// TwinCAT 3 PLC project PMPS
// Title: PMPS
// Company: SLAC - LCLS
// Author: Alex Wallace and contributors
// ProjectVersion: 0.0.0
// Description: Collection of PMPS functionality for LCLS PLCs
// ProgramVersion: 3.1.4023.0
// CompilerDefines: L
// libraries:
//   LCLS General, * (SLAC)
//   Tc2_MC2, * (Beckhoff Automation GmbH)
//   Tc2_Standard, * (Beckhoff Automation GmbH)
//   Tc2_System, * (Beckhoff Automation GmbH)
//   Tc2_Utilities, * (Beckhoff Automation GmbH)
//   Tc3_JsonXml, * (Beckhoff Automation GmbH)
//   Tc3_Module, * (Beckhoff Automation GmbH)
//   TcUnit,1.2.0.0,www.tcunit.org
// project tree:
//   AncillaryComponents/ FB_JsonDocToSafeBP.TcPOU, FB_JsonFileToJsonDoc.TcPOU, FB_TempSensor_FFO.TcPOU, FB_PressSensor_FFO.TcPOU
//   DUTs/InternalDUT/ E_MPSBeamRates.TcDUT, E_MPSBeamClasses.TcDUT, K_Apertures.TcDUT, K_Attenuators.TcDUT, K_Stopper.TcDUT, L_Apertures.TcDUT, L_Attenuators.TcDUT, L_Stopper.TcDUT, ST_AttenuatorStatus.TcDUT, ST_BP_ArbInternal.TcDUT, ST_FF.TcDUT, ST_FFInfo.TcDUT, ST_FFOverride.TcDUT, ST_PMPS_Aperture.TcDUT, ST_PMPS_Attenuator.TcDUT, T_HashTableEntry.TcDUT
//   DUTs/ PMPS_CODES.TcDUT, ST_DeviceState.TcDUT, ST_DeviceStateExt.TcDUT, ST_DeviceStateTable.TcDUT
//   DUTs/UserDUT/ E_BridgeLinkStatus.TcDUT, E_BridgeStatus.TcDUT, E_DataStatus.TcDUT, E_EcCommState.TcDUT, ST_ReactiveParams.TcDUT, ST_BeamParams.TcDUT, ST_DbStateParams.TcDUT, ST_Device.TcDUT
//   GVLs/ PMPS_GVL.TcGVL, PMPS_PARAM.TcGVL, PMPS_TOOLS.TcGVL
//   HelperFunctions/ FB_DummyHA.TcPOU, FB_DummyArbIO.TcPOU, F_BPWithID.TcPOU, F_DifferentBeamParams.TcPOU, F_eVExcludeRange.TcPOU, F_eVIncludeRange.TcPOU, F_eVRangeCalculator.TcPOU, F_eVWithinSpec.TcPOU, F_InitTestBP.TcPOU, F_SafeBPCompare.TcPOU, F_SafeBPCompare0Rate.TcPOU, F_SetBeamParams.TcPOU, F_SetGoodAttStatus.TcPOU, F_SetStateParams.TcPOU, F_PMPS_JSON.TcPOU, F_ValidReqID.TcPOU, PE_Ranges.TcPOU, F_AttenuatorOK.TcPOU
//   HelperFunctions/TypeTranslators/ APT_TO_IO.TcPOU, ATT_TO_IO.TcPOU, BP_TO_IO.TcPOU, F_DeviceState_To_DeviceStateExt.TcPOU, IO_TO_APT.TcPOU, IO_TO_ATT.TcPOU, IO_TO_BP.TcPOU
//   ImplicitChecks/ CheckBounds.TcPOU, CheckDivDInt.TcPOU, CheckDivLInt.TcPOU, CheckDivLReal.TcPOU, CheckDivReal.TcPOU, CheckLRangeSigned.TcPOU, CheckLRangeUnsigned.TcPOU, CheckPointer.TcPOU, CheckRangeSigned.TcPOU, CheckRangeUnsigned.TcPOU
//   / MAIN.TcPOU, PlcTask.TcTTO
//   MajorComponents/Arbiter/ FB_VetoArbiter.TcPOU, FB_Arbiter.TcPOU, FB_BeamParamAssertionPool.TcPOU
//   MajorComponents/BPTM/ BeamParameterTransitionManager.TcPOU, E_BPTMState.TcDUT
//   MajorComponents/ FB_BPControlDevice.TcPOU, FB_RateFromEPICS.TcPOU, FB_BeamClassFromEPICS.TcPOU, I_LowerAuthority.TcIO, I_UndulatorComplex.TcIO, FB_BPRequestor.TcPOU, FB_LinearDeviceStateTable.TcPOU, FB_LinearGovernor.TcPOU, I_HigherAuthority.TcIO
//   MajorComponents/PhotonEnergyInterface/ FB_AcceleratorLinks.TcPOU, FB_Hgvpu.TcPOU, FB_LPhotonEnergy.TcPOU, FB_KPhotonEnergy.TcPOU, FB_PhotonEnergy.TcPOU, FB_SXU.TcPOU, FB_UndulatorSegment.TcPOU, F_CalculatePhotonEnergy.TcPOU
//   MajorComponents/FastFaults/ FB_FastFault.TcPOU, FB_HardwareFFOutput.TcPOU
//   MajorComponents/InterPlcComm/ FB_ArbiterToSubSys_IO.TcPOU, FB_BridgeDiagnostics.TcPOU, FB_SubSysToArbiter_IO.TcPOU
//   MajorComponents/InterPlcComm/Sanitization/ I_FallibleLreal.TcIO, FB_FallibleRealFromEtherCAT.TcPOU
//   MajorComponents/PMPS_MPS_Interface/ FB_BeamClassOutputs.TcPOU, FB_BeamClassOutputs_BCD.TcPOU, FB_CTLS_Outputs.TcPOU, FB_MachineModeFromEPICS.TcPOU, FB_PhotonEnergyWatcher.TcPOU, FB_BeamClassWatcher.TcPOU
//   MajorComponents/SimulationFB/ FB_eVSimulator.TcPOU, FB_MachineSimulator.TcPOU
//   MajorComponents/Stoppers/ FB_KStopper.TcPOU, FB_KVetoDevice.TcPOU, FB_LVetoDevice.TcPOU, FB_LStopper.TcPOU, FB_StopperWatcher.TcPOU, FB_VetoDevice.TcPOU
//   TestComponents/DUT/ E_ArbDosTestStates.TcDUT, E_BPTMTestStates.TcDUT
//   TestComponents/ FB_Arbiter_Test.TcPOU, FB_VetoArbiter_Test.TcPOU, FB_AttenuatorSimulator.TcPOU, FB_BPTM_Test.TcPOU, FB_ArbToSubsys_Test.TcPOU, FB_DiffBP_Test.TcPOU, FB_SubsysToArb_Test.TcPOU, FB_evRangeCalculator_Test.TcPOU, FB_eVWithinSpec_Test.TcPOU, FB_FastFault_Test.TcPOU, FB_PhotonEnergyWatcher_Test.TcPOU, FB_SafeBPCompare_Test.TcPOU, FB_SolidAttenuator.TcPOU (excluded from build)
// real-time tasks:
//   TASK PlcTask: cycle T#10ms, priority 20, ADS port 350

CONFIGURATION PMPS
    RESOURCE PLC ON TwinCAT3
        TASK PlcTask(INTERVAL := T#10ms, PRIORITY := 20);
        PROGRAM MAIN WITH PlcTask : MAIN;
    END_RESOURCE
END_CONFIGURATION

// ---- DUTs/InternalDUT/E_MPSBeamRates.TcDUT

TYPE E_MPSBeamRates :
(
    MPSRateInvalid            :=  0,
    MPSRate0Hz                :=  1,
    (* Previously used 2 and 3 for single shot and burst *)
    MPSRate1Hz                :=  4,
    MPSRate10Hz               :=  5,
    MPSRate30Hz               :=  6,
    MPSRate60Hz               :=  7,
    MPSRate120Hz              :=  8,
    MPSRateUnknown            :=  9,
    MPSRateSingleShot         := 10,
    MPSRateBurstMode          := 11,
    MPSRateBurstModeNotActive := 12,
    MPSNumberOfBeamRates      := 13,
    MPSRateBurstInvalid       := 14
)UINT;
END_TYPE

// ---- DUTs/InternalDUT/E_MPSBeamClasses.TcDUT

TYPE E_MPSBeamClasses :
(
    Beam_Off    :=  0,
    Kicker_STBY :=  1,
    BC1Hz       :=  2,
    BC10Hz      :=  3,
    BC120Hz     :=  4,
    Diagnostic  :=  5,
    Tuning      :=  6,
    MAP_1       :=  7,
    MAP_5       :=  8,
    MAP_10      :=  9,
    MAP_25      := 10,
    MAP_50      := 11,
    MAP_100     := 12,
    FULL        := 13,
    SPARE1      := 14,
    SPARE2      := 15
);
END_TYPE

// ---- DUTs/InternalDUT/K_Apertures.TcDUT
{attribute 'qualified_only'}
{attribute 'strict'}
{attribute 'to_string'}
TYPE K_Apertures :
(
    SL1K0 := 1,
    SL2K0 := 2
);
END_TYPE

// ---- DUTs/InternalDUT/K_Attenuators.TcDUT
{attribute 'qualified_only'}
{attribute 'strict'}
TYPE K_Attenuators :
(
    AT1K0 := 1, // FEE Gas Attenuator
    AT1K4 := 2, // TMO Solid Attenuator in the FEE
    AT1K2 := 3, // RIX Solid Attenuator
    AT2K2 := 4, // RIX Solid Attenuator
    AT1K3 := 5 // TXI Solid Attenuator
);
END_TYPE

// ---- DUTs/InternalDUT/K_Stopper.TcDUT
{attribute 'qualified_only'}
{attribute 'strict'}
TYPE K_Stopper :
(
    ST3K4 := 1, // TMO PPS stopper in
    ST1K2 := 2, // RIX PPS stopper in
    MR1K1_IN := 3, // Monochromator focus optic vertical state
    MR1K1_OUT := 4, // Monochromator focus optic vertical state
    MR1K3_IN := 5, // TXI MR1K3 Offset Mirror horizontal state
    MR1K3_OUT := 6, // TXI MR1K3 Offset Mirror horizontal state
    ST4K4 := 7, //TMO ST4K4 Photon Terminator In Limit Switch
    ST1K0 := 8, //Test Photon Stopper in the FEE
    ST1K3 :=9, //TXI Kline PPS stopper in
    MR2K3_IN := 10, // TXI MR2K3 Offset Mirror state
    MR2K3_OUT := 11, // TXI MR2K3 Offset Mirror horizontal state
    DEFAULT := PMPS_GVL.MAX_VETO_DEVICES // DO NOT USE FOR ANYTHING
);
END_TYPE

// ---- DUTs/InternalDUT/L_Apertures.TcDUT
{attribute 'qualified_only'}
{attribute 'strict'}
{attribute 'to_string'}
TYPE L_Apertures :
(
    SL1L0 := 1,
    SL2L0 := 2
);
END_TYPE

// ---- DUTs/InternalDUT/L_Attenuators.TcDUT
{attribute 'qualified_only'}
{attribute 'strict'}
{attribute 'to_string'}
TYPE L_Attenuators :
(
    AT1L0 := 1, // FEE Combo Gas/Solid Attenuator
    AT2L0 := 2 // FEE Solid Attenuator
);
END_TYPE

// ---- DUTs/InternalDUT/L_Stopper.TcDUT
{attribute 'qualified_only'}
{attribute 'strict'}
TYPE L_Stopper :
(
    ST1L0 := 1, // ST1
    ST1L1 := 2, // TXI PPS Stopper in
    MR1L0_L0 := 3, // MR1L0 Pitch state delivery to L0 line
    MR1L0_TXI := 4, //MR1L0 Pitch state delivery to TXI line
    MR1L1_IN:= 5, //  TXI Offset Mirror horizontal state
    MR1L1_OUT:= 6, // TXI Offset Mirror horizontal state
    ST1L2 := 7, // ST1L2 XPP Stopper
    XPP_SB23_MONO:=8, // Indicates that XPP SB2/3 is in MONO Line
    XPP_SB23_PINK:=9, //Indicates that XPP SB2/3 is in PINK Line
    XPP_SB6_MONO:=10, // Indicates that XPP SB6is in MONO Line
    XPP_SB6_PINK:=11, //Indicates that XPP SB6 is in PINK Line
    ST2L0 := 12, // ST2L0 XRT Stopper
    DEFAULT := PMPS_GVL.MAX_VETO_DEVICES // DO NOT USE FOR ANYTHING
);
END_TYPE

// ---- DUTs/InternalDUT/ST_AttenuatorStatus.TcDUT
TYPE ST_AttenuatorStatus :
STRUCT
    AtTarget : BIT;     //0
    Moving : BIT;       //1
    LocalMode : BIT;    //2  (* means the attenuator ignores PMPS preemptive requests and operates from a local setpoint *)
    PMPSMode : BIT;     //3  (* means the attenuator is only taking setpoints from the pmps *)
    OK : BIT;           //4
    Toggle : BIT;       //5  just here for fun
    Include : BIT;      //6  Consider this device status
END_STRUCT
END_TYPE

// ---- DUTs/InternalDUT/ST_BP_ArbInternal.TcDUT
TYPE ST_BP_ArbInternal EXTENDS ST_BeamParams :
STRUCT
    {attribute 'pytmc' := 'pv: ID
        io: i
    '}
    nId : DWORD;
    {attribute 'pytmc' := 'pv: Live
        io: i
    '}
    LiveInTable : BOOL;
    {attribute 'pytmc' := 'pv: Device
        io: i
    '}
    sDevName: STRING;
END_STRUCT
END_TYPE

// ---- DUTs/InternalDUT/ST_FF.TcDUT
TYPE ST_FF :
STRUCT
    {attribute 'pytmc' := '
        pv: Info
     '}
    Info : ST_FFInfo;

    {attribute 'pytmc' := '
        pv: Ovrd
     '}
    Ovrd : ST_FFOverride;

    {attribute 'pytmc' := '
        pv: OK
        io: i
     '}
    OK   :   BOOL; // Fault logic state

    FaultAck : BOOL; // Set when faulted, reset by logger.
    ClearAck : BOOL;

    {attribute 'pytmc' := '
        pv: BeamPermitted
        io: i
     '}
    BeamPermitted   :   BOOL; // Result of reset, veto, and fault logic, true beam off boolean

    {attribute 'pytmc' := '
        pv: Reset
        io: o
     '}
    Reset   :   BOOL;

    bsFF    :    RS;
    rtReset    :    R_TRIG;
    ftCountFault : F_TRIG;

END_STRUCT
END_TYPE

// ---- DUTs/InternalDUT/ST_FFInfo.TcDUT

// These elements should be set at init and never changed.

TYPE ST_FFInfo :
STRUCT
    {attribute 'pytmc' := '
        pv: Path
        io: i
     '}
    sPath   :    T_MaxString; // Full PLC path to FF object
    {attribute 'pytmc' := '
        pv: Desc
        io: i
     '}
    Desc    :   T_MaxString; // Set at instantiation to a helpful description of the fast fault purpose
    {attribute 'pytmc' := '
        pv: DevName
        io: i
     '}
    DevName :   T_MaxString; // Component name, used in diagnostic to help narrow down where beam faults are coming from
    {attribute 'pytmc' := '
        pv: TypeCode
        io: i
     '}
    TypeCode    :   UINT; // Set at instantiation to fault class code

///////////////////////////////////////////
// Warning, this variable is effectively a VETO of the fast fault if set FALSE
// Do not alter the state of this variable unless you really know what you're doing.
///////////////////////////////////////////
    {attribute 'pytmc' := '
        pv: InUse
        io: i
     '}
    InUse   :   BOOL := FALSE; // If this FF is currently in-use
///////////////////////////////////////////


    AutoReset   :   BOOL; // Automatically clear fast fault (latching vs non-latching)
    Vetoable  : BOOL := TRUE; // Can this fast fault be masked by the veto device input?

      {attribute 'pytmc' := '
        pv: InfoString
        io: i
     '}
    InfoString : STRING;
END_STRUCT
END_TYPE

// ---- DUTs/InternalDUT/ST_FFOverride.TcDUT
TYPE ST_FFOverride :
STRUCT
    {attribute 'pytmc' := '
        pv: Duration
        io: o
     '}
    Duration : DINT; // DINT to be compatible with EPICS

    {attribute 'pytmc' := '
        pv: Expiration
        io: o
     '}
    Expiration : DINT; // DINT to be compatible with EPICS

    {attribute 'pytmc' := '
        pv: StartDT
        io: o
     '}
    StartDT : DINT; // DINT to be compatible with EPICS

    {attribute 'pytmc' := '
        pv: Activate
        io: o
     '}
    Activate : BOOL;

    {attribute 'pytmc' := '
        pv: Deactivate
        io: o
     '}
    Deactivate : BOOL;

    {attribute 'pytmc' := '
        pv: ElapsedTime
        io: i
     '}
    ElapsedTime : DINT; // DINT to be compatible with EPICS

    {attribute 'pytmc' := '
        pv: RemainingTime
        io: i
     '}
    RemainingTime : DINT; // DINT to be compatible with EPICS

    {attribute 'pytmc' := '
        pv: Active
        io: i
     '}
    Active: BOOL;

    Timer    :   TP;
    OvrdActLogAck : BOOL;
    OvrdExpLogAck : BOOL;

    tOvrdActivate : R_TRIG;
    tOvrdExpiring  : F_TRIG;
END_STRUCT
END_TYPE

// ---- DUTs/InternalDUT/ST_PMPS_Aperture.TcDUT
TYPE ST_PMPS_Aperture EXTENDS ST_PMPS_Aperture_IO :
STRUCT
    (*
    {attribute 'pytmc' := 'pv: Width
            io: i
            field: EGU mm'}
    Width : REAL; // distance between horizontal slits (x)
    {attribute 'pytmc' := 'pv: Height
            io: i
            field: EGU mm'}
    Height : REAL; // distance between vertical slits (y)

    {attribute 'pytmc' := 'pv: OK
        io: i'}
    xOK : BOOL; // status of aperture, false if error or in motion
    *)
END_STRUCT
END_TYPE

// ---- DUTs/InternalDUT/ST_PMPS_Attenuator.TcDUT
TYPE ST_PMPS_Attenuator EXTENDS ST_PMPS_Attenuator_IO :
STRUCT
    (*
        {attribute 'pytmc' := 'pv: Att
            io: i
            field: EGU %
        '}
        nTran : UINT;
        {attribute 'pytmc' := 'pv: OK
            io: i
        '}
        xAttOK : UINT; // true = no errors and attenuator is stable
        *)
END_STRUCT
END_TYPE

// ---- DUTs/InternalDUT/T_HashTableEntry.TcDUT
TYPE T_HashTableEntry :
STRUCT
    {attribute 'pytmc' := '
        pv: Key
        io: i
     '}
    key : DWORD := 0;
    value : PVOID := 0;
END_STRUCT
END_TYPE

// ---- DUTs/PMPS_CODES.TcDUT
{attribute 'qualified_only'}
{attribute 'strict'}
TYPE PMPS_CODES :
(
    FAST_FAULT := 16#1, // Generic fast fault
    PEW_FAULT := 16#7, // Fault occurs when the calculated machine photon energy (K value calculated by undulator gap, and electron energy) falls outside the permitted range.

    // Arbiter codes
    //////////////////////////////////
        ARB_FULL := 16#201, // Arbiter pool is full.

    //BPTM Codes
    //////////////////////////////////
        BadTargetID := 16#300,
        BadTransID := 16#301,
        TransAssrtFail := 16#302,
        FinalAssrtFail := 16#303,
        NoRoomInArb := 16#304
) UINT;
END_TYPE

// ---- DUTs/ST_DeviceState.TcDUT
TYPE ST_DeviceState :
STRUCT

    //State name
    sStateName	:	STRING;
    nStateRef	:	UDINT; //Primary key of device state database

    //////////////////
    // This stuff may belong in a sub-class or something
    //Position
    rPosition	:	REAL := 0; //Center of the state
    //Tolerance
    rTolerance :	REAL := 0; //+/- amount
    //////////////////
    //Required beam parameters
    stReqBeamParam	:	ST_BeamParams;

END_STRUCT
END_TYPE

// ---- DUTs/ST_DeviceStateExt.TcDUT
//Use when working with states in code
//Extended with a valid boolean to indicate the structure was loaded
//properly
TYPE ST_DeviceStateExt EXTENDS ST_DeviceState :
STRUCT
    xValid	:	BOOL := FALSE;
END_STRUCT
END_TYPE

// ---- DUTs/ST_DeviceStateTable.TcDUT
TYPE ST_DeviceStateTable :
STRUCT
    iDeviceID:DINT;
    iStateID:DINT;
    rTargetPosition: REAL;
    rTolerance: REAL;
    rTransmission: REAL;
    iBeamClass : DINT;
    iPulseRate: DINT;
    rPerPulseEnergy:REAL;
    rUpper_eV: REAL;
    rLower_eV: REAL;
    rPhotonEnergy: REAL;
END_STRUCT
END_TYPE

// ---- DUTs/UserDUT/E_BridgeLinkStatus.TcDUT
{attribute 'qualified_only'}
{attribute 'strict'}
{attribute 'to_string'}
TYPE E_BridgeLinkStatus :
(
    Connected,                    // local State = OP, far device present, far side TxPDOState = 0 (OP)
    LocalNotOperational,          // local State <> OP
    RemoteNotConnected,   // far device not present
    RemoteNotOperational          // far device present but TxPDOState <> 0
) UDINT;
END_TYPE

// ---- DUTs/UserDUT/E_BridgeStatus.TcDUT
{attribute 'qualified_only'}
{attribute 'strict'}
{attribute 'to_string'}
TYPE E_BridgeStatus :
(
    Connected,
    LocalNotOperational,
    RemoteNotConnected,
    RemoteNotOperational,
    LinkError,
    DataStale
) UDINT;
END_TYPE

// ---- DUTs/UserDUT/E_DataStatus.TcDUT
{attribute 'qualified_only'}
{attribute 'strict'}
{attribute 'to_string'}
TYPE E_DataStatus :
(
    Ok,
    WcError,   // working counter reports invalid data
    Stale      // WC valid but the input toggle hasn't changed for the timeout window
) UDINT;
END_TYPE

// ---- DUTs/UserDUT/E_EcCommState.TcDUT
TYPE E_EcCommState : (
    eEcState_UNDEFINED 	:= 0,
    eEcState_INIT 		:= 1,
    eEcState_PREOP 		:= 2,
    eEcState_BOOT 		:= 3,
    eEcState_SAFEOP 	:= 4,
    eEcState_OP 		:= 8
) UDINT;
END_TYPE

// ---- DUTs/UserDUT/ST_ReactiveParams.TcDUT
TYPE ST_ReactiveParams :
STRUCT
    {attribute 'pytmc' := 'pv: TempSP
            io: i
            field: PREC 2;
            field: EGU "C";
        '}
    nTempSP: REAL;
    {attribute 'pytmc' := 'pv: PressSP
            io: i
            field: PREC 2;
            field: EGU "TORR";
        '}
    nPressSP: REAL;
END_STRUCT
END_TYPE

// ---- DUTs/UserDUT/ST_BeamParams.TcDUT
TYPE ST_BeamParams :
    STRUCT
        (*  Requested pre-optic attenuation %  *)
        {attribute 'pytmc' := 'pv: Transmission
            io: i
            field: HOPR 1;
            field: LOPR 0;
            field: PREC 2;
        '}
        nTran : REAL := 0;
        (* Pulse-rate *)
        {attribute 'pytmc' := 'pv: Rate
            io: i
            field: EGU Hz
        '}
        nRate : UDINT := 0;
        (* Photon energy ranges *)
        {attribute 'pytmc' := 'pv: eVRanges
            io: i
            field: EGU eV'}
        {attribute 'displaymode' := 'binary'}
        neVRange : DWORD := 0;
                 (* Photon energy  *)
        {attribute 'pytmc' := 'pv: PhotonEnergy
            io: i
            field: EGU eV'}
        neV : REAL := 0;
        (* Beamclass ranges *)
         {attribute 'pytmc' := 'pv: BeamClassRanges
            io: i'}
        {attribute 'displaymode' := 'binary'}
        nBCRange : WORD := 0;
        (* Beamclass *)
        {attribute 'pytmc' := 'pv: BeamClass
            io: i'}
        nBeamClass : USINT :=0;
        (* Machine Mode *)
        {attribute 'pytmc' := 'pv: MachineMode
            io: i'}
        nMachineMode: USINT:=3;
        (* Beamline attenuators *)
        {attribute 'pytmc' := 'pv: AuxAtt
        io: i'}
        astAttenuators : ARRAY [1..PMPS_GVL.AUX_ATTENUATORS] OF ST_PMPS_Attenuator;

        (* Stoppers *)
        {attribute 'pytmc' := 'pv: Veto
        io: i'}
        aVetoDevices : ARRAY [1..PMPS_GVL.MAX_VETO_DEVICES] OF BOOL;

        (* Apertures *)
        {attribute 'pytmc' := 'pv: Apt
        io: i'}
        astApertures : ARRAY [1..PMPS_GVL.MAX_APERTURES] OF ST_PMPS_Aperture := [(Width:=1E3, Height:=1E3), (Width:=1E3, Height:=1E3),(Width:=1E3, Height:=1E3),(Width:=1E3, Height:=1E3)];

        // Toggle for watchdog
        xValidToggle : BOOL;
        // Beam parameter set is valid (if readback), or acknowledged (if request)
        {attribute 'pytmc' := 'pv: Valid
        io: i'}
        xValid : BOOL;
        // Cohort index. Identifies which cohort this BP set was included in arbitration
        {attribute 'pytmc' := 'pv: Cohort
        io: i
            field: DESC Cohort inc on each arb cycle
        '}
        nCohortInt : UDINT;
    END_STRUCT
END_TYPE

// ---- DUTs/UserDUT/ST_DbStateParams.TcDUT
TYPE ST_DbStateParams :
     // Defines The parameters that are loaded from the json db for every state name
STRUCT
      // PMPS database lookup name for this state
    {attribute 'pytmc' := '
        pv: PMPS_STATE
        io: i
        field: DESC PMPS Database Lookup Key
    '}
    sPmpsState: STRING;

    // Beam parameters associated with this state
    {attribute 'pytmc' := '
        pv: BP
        io: i
    '}
    stBeamParams: ST_BeamParams := PMPS_GVL.cst0RateBeam;

    // Set to TRUE once the PMPS library has loaded a valid state from the database
    {attribute 'pytmc' := '
        pv: PMPS_LOADED
        io: i
        field: DESC TRUE if PMPS loaded parameters from the database.
    '}
    bBeamParamsLoaded: BOOL;

     // Reactive parameters associated with this state
    {attribute 'pytmc' := '
        pv: ReParams
        io: i
    '}
    stReactiveParams : ST_ReactiveParams;

    // Transition ID associated with this state
    {attribute 'pytmc' := '
        pv: PMPS_ID
        io: i
        field: DESC Assertion Request ID
    '}
    nRequestAssertionID: UDINT;
END_STRUCT
END_TYPE

// ---- DUTs/UserDUT/ST_Device.TcDUT
TYPE ST_Device :
STRUCT
    //IO
    stAxis	:	AXIS_REF;
    //The following limit switches must be TRUE or high (ie. NC) to enable that direction of motion
    //The EPICS display should show an inverted indicator to communicate end of travel reached
    i_xLoLim	AT %I*	:	BOOL; //Wire normally-closed
    i_xHiLim	AT %I*	:	BOOL; //Wire normally-closed

    //Acuator Parameters
    lrUpperPositionLimit	:	LREAL := 10000000000; //Use in conjuntion with limit switches or set to a huge number to ignore
    lrLowerPositionLimit	:	LREAL := -10000000000; //Use in conjuntion with limit switches or set to a huge number to ignore

    xEnable	:	BOOL := TRUE;

    //Supervisory System

    //MPS Override
    xOverrideMPSLimits	: BOOL := FALSE; //Set true to move beyond MPS limits. Note this will trip beam off.

    //Status and Faults
    xClearFaults	:	BOOL;	//Rising edge tries to clear faults of all kinds

    xGovernorFault	:	BOOL;	//Indicates governor is faulted
    xGovernorOverridden	:	BOOL; //Indicates governor is in override mode
    xSMFault		:	BOOL;	//Indicates component state machine is faulted

    //Device States
    StateTable		:	FB_LinearDeviceStateTable;

    stTransitionState	:	ST_DeviceState; //The transition state might have non-zero beam parameters
    nSafeState			:	UDINT; //State where the device is considered safe
    nTransitionState	:	UDINT;

    nRequestedState	:	UDINT; //EPICS control, cleaned (checked against array limits) and deposited in nTargetState
    nTargetState	:	UDINT; //The requested state should be deposited here after cleaning
    nActiveState	:	UDINT; //The last successfully reached state


END_STRUCT
END_TYPE

// ---- MajorComponents/BPTM/E_BPTMState.TcDUT
TYPE E_BPTMState :
(
    Init := 0,
    NewTarget := 1000,
    RequestBP := 1500,
    WaitForBP := 2500,
    WaitingForTransitionAssertion := 2000,
    WaitingForFinalAssertion := 3000,
    Transitioning := 4000,
    WaitForFinalBP := 5000,
    CleaningUp := 6000,
    Idle := 10000,
    Done := 8000,
    Error := 9000
);
END_TYPE

// ---- TestComponents/DUT/E_ArbDosTestStates.TcDUT
{attribute 'qualified_only'}
{attribute 'strict'}
TYPE E_ArbDosTestStates :
(
    Init := 0,
    SecondReq := 100,
    WaitForAck := 200,
    WaitFor2ndAck := 300,
    RunAsserts := 8000
);
END_TYPE

// ---- TestComponents/DUT/E_BPTMTestStates.TcDUT
{attribute 'qualified_only'}
{attribute 'strict'}
TYPE E_BPTMTestStates :
(
    Init := 0,
    WaitingForValidID := 50,
    WaitingForTransitionAssertion := 100,
    StalledAtTransition := 150,
    WaitingForFinalAssertion    := 200,
    WaitingForBeam := 250,
    Transitioning    := 300,
    CleaningUp    := 400,
    AnotherState := 500,
    Retry := 1000,
    Done := 8000,
    Error := 9000
);
END_TYPE

// ---- GVLs/PMPS_GVL.TcGVL
{attribute 'qualified_only'}
VAR_GLOBAL
    {attribute 'pytmc' := '
        pv: @(PREFIX)RequestedBP
        io: i
        archive: 1Hz monitor
    '}
    stRequestedBeamParameters    :    ST_BeamParams; //Summarized request for the line, as recognized by the line arbiter PLC
    {attribute 'pytmc' := '
        pv: @(PREFIX)CurrentBP
        io: i
        archive: 1Hz monitor
    '}
    stCurrentBeamParameters    :    ST_BeamParams; //Currently active BP set, broadcast by the line arbiter PLC

    {attribute 'pytmc' := '
        pv: @(PREFIX)eVRangeCnst
        io: i
        archive: 1Hz monitor
        field: DESC Active eV Range constants
        field: EGU eV
    '}
    g_areVBoundaries    :    ARRAY [0..g_cBoundaries]    OF    REAL;



    PERange : PE_Ranges; //Included to place the ev ranges properly
END_VAR
VAR_GLOBAL RETAIN
    // Statistics
    {attribute 'pytmc' := '
        pv: @(PREFIX)SuccessfulPreemptions
        io: i
    '}
    SuccessfulPreemption : UDINT; // Any time BPTM applies a new BP request which is confirmed
    {attribute 'pytmc' := '
        pv: @(PREFIX)AccumulatedFastFaults
        io: i
    '}
    AccumulatedFF : UDINT; // Any time a FF occurs
    BP_jsonDoc 		: SJsonValue;
END_VAR
VAR_GLOBAL CONSTANT

    EXCLUDED_ASSERTION_ID    :    UDINT    := 16#FFFFFFFF; //An assertion ID that should always return "not found" in the assertion pool
    VISIBLE_TEST_VELOCITY    :    LREAL    := 10;
    FAST_TEST_VELOCITY        :    LREAL    := 100;
    MAX_DEVICE_STATES        :    UDINT    := 300;

    TRANS_SCALING_FACTOR : REAL := REAL#1.0; // Scaling factor for fixed-point transmission

    AUX_ATTENUATORS : UINT := 16; // Maximum # of attenuators in the PMPS
    MAX_VETO_DEVICES   :   UINT := 16;
    stAttenuators : ST_PMPS_Attenuator :=(nTran:=1,xAttOK:=1);
    {attribute 'pytmc' := '
        pv: @(PREFIX)FullBeamCnst
        io: i
        archive: 1Hz monitor
        field: DESC Full beam constant
    '}
    cstFullBeam    :    ST_BeamParams := (
        nTran := 1,
        neVRange :=  2#1111_1111_1111_1111_1111_1111_1111_1111,
        nRate    := UDINT#1000000,
        nBCRange := 2#0111_1111_1111_1111,
        astApertures := [(Width:=1E3, Height:=1E3), (Width:=1E3, Height:=1E3),(Width:=1E3, Height:=1E3),(Width:=1E3, Height:=1E3)],
        astAttenuators :=  [PMPS_GVL.AUX_ATTENUATORS(stAttenuators)]

    );
    {attribute 'pytmc' := '
        pv: @(PREFIX)0RateBeamCnst
        io: i
        archive: 1Hz monitor
        field: DESC 0-rate beam constant
    '}
    cst0RateBeam    :    ST_BeamParams := ( // Use for transition requests
        nTran := 1,
        neVRange :=  2#1111_1111_1111_1111_1111_1111_1111_1111,
        nRate    := 0,
        nBCRange := 2#0000_0000_0000_0000,
        astApertures := [(Width:=1E3, Height:=1E3), (Width:=1E3, Height:=1E3),(Width:=1E3, Height:=1E3),(Width:=1E3, Height:=1E3)],
        astAttenuators :=  [PMPS_GVL.AUX_ATTENUATORS(stAttenuators)]
    );
   (*  {attribute 'pytmc' := '
        pv: @(PREFIX)SafeBeamCnst
        io: i
        archive: 1Hz monitor
        field: DESC Safe beam constant
    '}
   cstSafeBeam    :    ST_BeamParams := (
        nTran := 0,
        neVRange := 0,
        nRate    := 0
    );*)

    cnMaxStateArrayLen : INT := 20;


    MAX_APERTURES : UINT := 4; // Maximum # of power slits in the PMPS
    {warning disable C0228}
    DUMMY_AUX_ATT_ARRAY : ARRAY [1..PMPS_GVL.AUX_ATTENUATORS] OF ST_PMPS_Attenuator;
    {warning restore C0228}



    g_cBoundaries    :    INT    := 31;


//////////////////////////
// L Undulator constants
//////////////////////////

///////////////////////////////////////

    {attribute 'pytmc' := '
        pv: @(PREFIX)eVRangeHyst
        io: i
        archive: 1Hz monitor
        field: DESC eV Range hystersis
        field: EGU eV
    '}
    reVHyst: REAL := 5; //


    {attribute 'pytmc' := '
        pv: @(PREFIX)L:eVRangeCnst
        io: i
        archive: 1Hz monitor
        field: DESC eV Range constants
        field: EGU eV
    '}
    g_areVBoundariesL    :    ARRAY [0..g_cBoundaries]    OF    REAL    := [
    1.0E3,
    1.7E3,
    2.1E3,
    2.5E3,
    3.8E3,
    4.0E3,
    5.0E3,
    7.0E3,
    7.5E3,
    7.7E3,
    8.9E3,
    10.0E3,
    11.1E3,
    12.0E3,
    13.0E3,
    13.5E3,
    14.0E3,
    16.9E3,
    18.0E3,
    20.0E3,
    22.0E3,
    24.0E3,
    25.0E3,
    25.5E3,
    26.0E3,
    27.0E3,
    28.0E3,
    28.5E3,
    29.0E3,
    30.0E3,
    60.0E3,
    90.0E3
    ];


    {attribute 'pytmc' := '
        pv: @(PREFIX)K:eVRangeCnst
        io: i
        archive: 1Hz monitor
        field: DESC eV Range constants
        field: EGU eV
    '}
    g_areVBoundariesK    :    ARRAY [0..g_cBoundaries]    OF    REAL    := [
    100,
    250,
    270,
    350,
    400,
    450,
    480,
    530,
    680,
    730,
    850,
    1.10E3,
    1.15E3,
    1.25E3,
    1.45E3,
    1.50E3,
    1.55E3,
    1.65E3,
    1.70E3,
    1.75E3,
    1.82E3,
    1.85E3,
    2.00E3,
    2.20E3,
    2.50E3,
    2.80E3,
    3.00E3,
    3.15E3,
    3.50E3,
    4.00E3,
    5.30E3,
    7.00E3
    ];

    L_Stopper_Pairings : ARRAY[1..PMPS_GVL.MAX_VETO_DEVICES] OF L_STOPPER :=
    [
    L_Stopper.DEFAULT,		// L_Stopper.ST1L0
    L_Stopper.DEFAULT, 		// L_Stopper.ST1L1
    L_Stopper.MR1L0_TXI, 	// L_Stopper.MR1L0_L0
    L_Stopper.MR1L0_L0, 	// L_Stopper.MR1L0_TXI
    L_Stopper.MR1L1_OUT,	// L_Stopper.MR1L1_IN
    L_Stopper.MR1L1_IN  	// L_Stopper.MR1L1_OUT
    ];

    K_Stopper_Pairings : ARRAY[1..PMPS_GVL.MAX_VETO_DEVICES] OF K_STOPPER :=
    [
    K_Stopper.DEFAULT,		// ST3K4
    K_Stopper.DEFAULT,		// ST1K2
    K_Stopper.MR1K1_OUT,	// MR1K1_IN
    K_Stopper.MR1K1_IN,		// MR1K1_OUT
    K_Stopper.MR1K3_OUT,	// MR1K3_IN
    K_Stopper.MR1K3_IN,		// MR1K3_OUT
    K_Stopper.DEFAULT,		// ST4K4
    K_Stopper.DEFAULT,		// ST1K4
    K_Stopper.DEFAULT,		// ST1K3
    K_Stopper.MR2K3_OUT,	// MR2K3_IN
    K_Stopper.MR2K3_IN		// MR2K3_OUT
    ];

END_VAR

// ---- GVLs/PMPS_PARAM.TcGVL
{attribute 'qualified_only'}
VAR_GLOBAL CONSTANT
    MAX_FAST_FAULTS	:	UINT := 50; // Max fast faults for an FFO
    MAX_ASSERTIONS    :    UDINT := 20; //Maximum number of BP requests in the arbiter
    TRANS_MARGIN : REAL := REAL#0.20; // Allowed % margin above requested transmission level in SafeBPCompare (0.2000 = 20deci% default). Note: change this value if scaling factor changes.
END_VAR

// ---- GVLs/PMPS_TOOLS.TcGVL
{attribute 'qualified_only'}
VAR_GLOBAL
    fbJson : FB_JsonSaxWriter;
END_VAR

// ---- MajorComponents/I_LowerAuthority.TcIO
INTERFACE I_LowerAuthority

PROPERTY bLowerAuthorityVetoed : BOOL
GET
END_GET
SET
END_SET
END_PROPERTY

// <Arbiter Internal>
// Elevates the arbitrated BP set to something above.
// Could be another arbiter, or a BP requester/ IO, 
// or an FB that locks in a specific portion of the BP set.
METHOD ElevateRequest : BOOL 
VAR_INPUT
    HigherAuthority : I_HigherAuthority;
END_VAR
END_METHOD

PROPERTY nLowerAuthorityID : DWORD
GET
END_GET
END_PROPERTY

END_INTERFACE

// ---- MajorComponents/I_UndulatorComplex.TcIO
INTERFACE I_UndulatorComplex

PROPERTY rCurrentPhotonEnergy : LREAL
GET
END_GET
END_PROPERTY

PROPERTY rTargetPhotonEnergy : LREAL
GET
END_GET
END_PROPERTY

END_INTERFACE

// ---- MajorComponents/InterPlcComm/Sanitization/I_FallibleLreal.TcIO

INTERFACE I_FallibleLreal


PROPERTY Error : BOOL
GET
END_GET
END_PROPERTY


PROPERTY Value : LREAL
GET
END_GET
END_PROPERTY

END_INTERFACE

// ---- MajorComponents/I_HigherAuthority.TcIO
INTERFACE I_HigherAuthority

//Verify with this higher authority that the request is being included
METHOD CheckRequest : BOOL
VAR_INPUT
    nReqID    :    DWORD;
END_VAR
END_METHOD

//Remove the request from this higher authority
METHOD RemoveRequest : BOOL
VAR_INPUT
	nReqID    :    DWORD; //StateID to remove
END_VAR
END_METHOD

// Request a BP from this higher authority
METHOD RequestBP : BOOL
VAR_INPUT
    nReqID    :    DWORD; //StateID of state requesting beam parameter set
    stReqBP        :    ST_BeamParams; //Requested beam params
END_VAR
END_METHOD

END_INTERFACE

// ---- MAIN.TcPOU
PROGRAM MAIN
VAR
    fbSetPERanges : PE_Ranges;

    fbDiffBPTest    :    FB_DiffBP_Test;
    fbBPTMTest    :    FB_BPTM_Test;
    fbSafeBPCompareTest    :    FB_SafeBPCompare_Test;
    ////fbevWithinSpecTest    :    FB_evWithinSpec_Test;---
    ////fbPEWTest    :    FB_PhotonEnergyWatcher_Test;---
    fbFFTest    :    FB_FastFault_Test;
    fbArbiterTest    :    FB_Arbiter_Test;
    fbVetoArbiterTest : FB_VetoArbiter_Test;
    fbevRangeCalcTest : FB_evRangeCalculator_Test;
    fbSubSysToArbTest : FB_SubsysToArb_Test;
    fbArbToSubSysTest : FB_ArbToSubsys_Test;
END_VAR

TcUnit.RUN();

END_PROGRAM

// ---- HelperFunctions/PE_Ranges.TcPOU
// Does nothing other than set the gvl for photon energy bitmask to one of two constants, K or L.
// Workaround for compile defines not fully working for libraries at the time of writing this.
// Otherwise I would have just used the compile define in the GVL declaration.
FUNCTION_BLOCK PE_Ranges
VAR_INPUT
END_VAR
VAR_OUTPUT
END_VAR
VAR
END_VAR

METHOD FB_init : BOOL
VAR_INPUT
    bInitRetains : BOOL; // if TRUE, the retain variables are initialized (warm start / cold start)
    bInCopyCode : BOOL;  // if TRUE, the instance afterwards gets moved into the copy code (online change)
END_VAR
{IF defined (L)}
    PMPS_GVL.g_areVBoundaries := PMPS_GVL.g_areVBoundariesL;
{ELSIF defined (K)}
    PMPS_GVL.g_areVBoundaries := PMPS_GVL.g_areVBoundariesK;
{END_IF}
END_METHOD

END_FUNCTION_BLOCK

// ---- TestComponents/FB_DiffBP_Test.TcPOU
{attribute 'call_after_init'}
FUNCTION_BLOCK FB_DiffBP_Test EXTENDS TcUnit.FB_TestSuite
VAR_INPUT
END_VAR
VAR_OUTPUT
END_VAR
VAR

END_VAR


BPDiff();

//Verify BP comparison remains logical.
METHOD BPDiff
VAR_INPUT
END_VAR
VAR
    BP1    :    ST_BeamParams;
    BP2    :    ST_BeamParams;
END_VAR
TEST('BPDiffCheck');

BP2.nTran := 10;

AssertTrue(
    F_DifferentBeamParams(BP1, BP2),
    'DifferentBP eval is broken (True)');

BP1.nTran := BP2.nTran;

AssertFalse(
    F_DifferentBeamParams(BP2, BP1),
    'DifferentBP eval is broken (False)');

TEST_FINISHED();
END_METHOD

END_FUNCTION_BLOCK

// ---- HelperFunctions/F_DifferentBeamParams.TcPOU
(*Compares BeamParam1 to BeamParam2, if any parameters of BeamParam1 are different than BeamParam2
the result will be true. *)
{attribute 'no_check'}
FUNCTION F_DifferentBeamParams : BOOL
VAR_INPUT
    BeamParam1    :    ST_BeamParams;
    BeamParam2    :    ST_BeamParams;
END_VAR
VAR
    xAttOK: BOOL := FALSE;
    xEvOK: BOOL := FALSE;
    xRateOK: BOOL := FALSE;
    xaStopper : BOOL := FALSE;
    xaAtt : BOOL := FALSE;
    xaApt : BOOL := FALSE;
    xBCOK : BOOL := FALSE;

    idx : UINT;


END_VAR

xAttOK := BeamParam1.nTran <> BeamParam2.nTran;
xEvOK := BeamParam1.neVRange <> BeamParam2.neVRange;
xRateOK     := BeamParam1.nRate <> BeamParam2.nRate;
xBCOK	:= BeamParam1.nBCRange <> BeamParam2.nBCRange;// OR BeamParam1.nBeamClass <> BeamParam2.nBeamClass ; //Is this right?


//ast Attenuators
FOR idx:=1 TO PMPS_GVL.AUX_ATTENUATORS DO
    xaAtt S= (BeamParam1.astAttenuators[idx].nTran <> BeamParam2.astAttenuators[idx].nTran);
END_FOR

// Stoppers
FOR idx:=1 TO PMPS_GVL.MAX_VETO_DEVICES DO
    xaStopper S= (BeamParam1.aVetoDevices[idx] <> BeamParam2.aVetoDevices[idx]);
END_FOR

// ast Apertures
FOR idx:=1 TO PMPS_GVL.MAX_APERTURES DO
    xaApt S= (BeamParam1.astApertures[idx].Height <> BeamParam2.astApertures[idx].Height) OR
            (BeamParam1.astApertures[idx].Width <> BeamParam2.astApertures[idx].Width);
END_FOR


F_DifferentBeamParams := xAttOK OR xEvOK OR xRateOK OR xaStopper OR xaAtt OR xaApt OR xBCOK;

END_FUNCTION

// ---- TestComponents/FB_BPTM_Test.TcPOU
{attribute 'call_after_init'}
FUNCTION_BLOCK FB_BPTM_Test EXTENDS TcUnit.FB_TestSuite
VAR_INPUT
END_VAR
VAR_OUTPUT
END_VAR
VAR
END_VAR
VAR CONSTANT
    BPTM_ARR : UDINT := PMPS_PARAM.MAX_ASSERTIONS;
    cCycle : UINT := 20; // How many cycles does it take to complete a BPTM
END_VAR

BPTMBasicFunction();
InterruptAtAllSteps();
FullArbError();

METHOD BPTMBasicFunction
VAR_INPUT
END_VAR
VAR
    //Final and transition assertions
    nTransitionID    :    UDINT := 1;
    stTransitionAssertion    :    ST_BeamParams := (nRate := 10, nBCRange:=0);

    nReqID    :    UDINT    := 2;
    stReqAssertion    :    ST_BeamParams := (nTran := 0.2, nBCRange:=2#0000_0000_0000_0011);

END_VAR
VAR_INST
    fbBPTM_TestBasicFunction    :    BeamParameterTransitionManager;
    fbArbiter    :    FB_Arbiter(1);
    ffo : FB_HardwareFFOutput;
    fbSubSysIO : FB_DummyArbIO;
    xFirstPass    :    BOOL := TRUE;
    eTestStep: E_BPTMTestStates := E_BPTMTestStates.Init;
END_VAR

// Completes arbiter request elevation process
// Necessary for CheckRequest to return true, ever
    fbBPTM_TestBasicFunction(
        fbArbiter := fbArbiter,
        );

fbSubSysIO(LA := fbArbiter, FFO := ffo);

// Note: this struct may also be (over)written to in the tests below, specifically rate.
fbBPTM_TestBasicFunction.stCurrentBeamParameters := fbSubSysIO.q_stSimulatedBPReadback;

//MG: Need to set the Machine mode testing SC
PMPS_GVL.stCurrentBeamParameters.nMachineMode :=0;

CASE eTestStep OF

E_BPTMTestStates.Init:

    TEST('BPTMTest');
    eTestStep := E_BPTMTestStates.WaitingForBeam;

E_BPTMTestStates.WaitingForBeam:
    TEST('BPTM Waits for Beam');

    fbBPTM_TestBasicFunction.i_TransitionAssertionID := nTransitionID;
    fbBPTM_TestBasicFunction.i_stTransitionAssertion := stTransitionAssertion;

    fbBPTM_TestBasicFunction.i_nRequestedAssertionID := nReqID;
    fbBPTM_TestBasicFunction.i_stRequestedAssertion := stReqAssertion;

    IF fbBPTM_TestBasicFunction.eBPTMState = E_BPTMState.WaitForBP AND
        NOT fbBPTM_TestBasicFunction.xEntry THEN

        AssertTrue(fbArbiter.CheckRequestInPool(nTransitionID), 'Arbiter did not accept BPTM transition assertion');

        AssertTrue(fbArbiter.CheckRequestInPool(nReqID), 'Arbiter did not accept BPTM transition assertion');

        AssertFalse(fbBPTM_TestBasicFunction.q_xTransitionAuthorized,
            'Transition should not be authorized until requests are in and beam is ready');

        AssertTrue(fbBPTM_TestBasicFunction.bBusy, 'Busy should be true here');
        AssertFalse(fbBPTM_TestBasicFunction.bDone, 'Done should be false');
        AssertFalse(fbBPTM_TestBasicFunction.bError, 'Error should be false here');

        TEST_FINISHED_NAMED('BPTM Waits for Beam');

        eTestStep := E_BPTMTestStates.Transitioning;
    END_IF


E_BPTMTestStates.Transitioning:
    TEST('BPTM Authorizes Transition');

    fbBPTM_TestBasicFunction.stCurrentBeamParameters.nRate := 0; // satisfies the transition request
    fbBPTM_TestBasicFunction.stCurrentBeamParameters.nBeamClass := 0; // satisfies the transition request

    IF fbBPTM_TestBasicFunction.eBPTMState = E_BPTMState.Transitioning AND
        NOT fbBPTM_TestBasicFunction.xEntry THEN

        AssertTrue(fbArbiter.CheckRequest(nTransitionID),
            'Transition assertion should be in arbiter');

        AssertTrue(fbArbiter.CheckRequest(nReqID),
            'Final assertion should be in arbiter');

        AssertTrue(fbBPTM_TestBasicFunction.q_xTransitionAuthorized,
            'Transition should be authorized at this point.');

        AssertEquals(nReqID, fbBPTM_TestBasicFunction.nCurrentAssertionID,
            'nCurrentAssertionID not set.');

        TEST_FINISHED_NAMED('BPTM Authorizes Transition');

        eTestStep := E_BPTMTestStates.WaitingForFinalAssertion;
    END_IF

E_BPTMTestStates.WaitingForFinalAssertion:
    TEST('BPTM Waits for final BP');

    fbBPTM_TestBasicFunction.i_xDoneMoving := TRUE;

    IF fbBPTM_TestBasicFunction.eBPTMState = E_BPTMState.WaitForFinalBP THEN

        AssertTrue(fbArbiter.CheckRequest(nTransitionID),
        'Transition assertion should be in arbiter');

        TEST_FINISHED_NAMED('BPTM Waits for final BP');

        eTestStep := E_BPTMTestStates.CleaningUp;
    END_IF

E_BPTMTestStates.CleaningUp:

    fbSubSysIO.AutoUpdateBP := TRUE;

    TEST('Cleaning up');

    IF fbBPTM_TestBasicFunction.eBPTMState = E_BPTMState.Done THEN

        AssertFalse(fbArbiter.CheckRequestInPool(nTransitionID), 'Transition req should be removed from arb now');

        eTestStep := E_BPTMTestStates.Done;

        TEST_FINISHED_NAMED('Cleaning up');
    END_IF

E_BPTMTestStates.Done:


    AssertTrue(fbBPTM_TestBasicFunction.bDone, 'Done should be set');
    AssertFalse(fbBPTM_TestBasicFunction.bError, 'Error should be cleared');
    AssertFalse(fbBPTM_TestBasicFunction.bBusy, 'Busy should be false');

    TEST_FINISHED_NAMED('BPTMTest');

END_CASE
END_METHOD

// Simulate error due to full arbiter
METHOD FullArbError
VAR_INPUT
END_VAR
VAR
    //Final and transition assertions
    nTransitionID    :    UDINT := 1000;
    stTransitionAssertion    :    ST_BeamParams :=  ( nTran := 0, neVRange := 0, nRate  := 0);//PMPS_GVL.cstSafeBeam;

    nReqID    :    UDINT    := 2000;
    stReqAssertion    :    ST_BeamParams := ( nTran := 0, neVRange := 0, nRate  := 0);//PMPS_GVL.cstSafeBeam;

    idx : UDINT;

    nRandID : DWORD;
    testReq : ST_BeamParams := (neVRange := 16#FFEE, nRate:=33);

END_VAR
VAR_INST
    fbBPTM_TestFullArb    :    BeamParameterTransitionManager;
    fbArbFullErr    :    FB_Arbiter(1);
    ffo : FB_HardwareFFOutput;
    fbSubSysIO : FB_DummyArbIO;
    fbBPR :  FB_BPRequestor;
    xFirstPass    :    BOOL := TRUE;
    eTestStep: E_BPTMTestStates := E_BPTMTestStates.Init;
    tonRetryTimeout : TON := (PT:=T#5s);
    entryToRetry : bool := true;
    fbRand : DRAND := (Seed :=1);
END_VAR
CASE eTestStep OF

E_BPTMTestStates.Init:

    TEST('BPTMErrorFullArb');

    // Fill the arbiter
    FOR idx := 1 TO PMPS_PARAM.MAX_ASSERTIONS // this fills the arbiter
                    - fbBPTM_TestFullArb.cReqArbCapacity + 1 DO // but test just one over the allowed amount
        fbArbFullErr.AddRequest(nReqID := idx, stReqBP := testReq, sDevName :='Device');
    END_FOR

    fbSubSysIO.AutoUpdateBP := TRUE;

    AssertTrue(PMPS_PARAM.MAX_ASSERTIONS - fbArbFullErr.nEntryCount < fbBPTM_TestFullArb.cReqArbCapacity,
        'Arbiter is not full enough, rest of tests will be invalid');

    eTestStep := E_BPTMTestStates.Error;

E_BPTMTestStates.Error:

    TEST('BPTM Full Error');

    IF fbBPTM_TestFullArb.bError THEN

        AssertTrue(fbBPTM_TestFullArb.bError AND fbBPTM_TestFullArb.nErrId = PMPS_CODES.NoRoomInArb,
            'Incorrect error response from full arbiter.');

        TEST_FINISHED_NAMED('BPTM Full Error');

        eTestStep := E_BPTMTestStates.Retry;

    END_IF

E_BPTMTestStates.Retry:

    TEST('Test Retry Post Failed Final');

    // Clear the arbiter
    if entryToRetry THEN
        FOR idx := 1 TO PMPS_PARAM.MAX_ASSERTIONS + 1 DO
            fbArbFullErr.RemoveRequest(idx);
        END_FOR
        entryToRetry := FALSE;
    END_IF

    // Push the retry button
    fbBPTM_TestFullArb.bRetry := TRUE;

    tonRetryTimeout(IN:=TRUE);

    IF tonRetryTimeout.Q OR fbBPTM_TestFullArb.q_xTransitionAuthorized THEN
        AssertTrue(fbBPTM_TestFullArb.q_xTransitionAuthorized, 'Transition should have been authorized by now');
        AssertTrue(fbArbFullErr.CheckRequest(nTransitionID), 'Transition ID is missing from arbiter while transition is authorized');
        AssertTrue(fbArbFullErr.CheckRequest(nReqID), 'Final ID is missing from arbiter while transition is authorized');

        TEST_FINISHED_NAMED('Test Retry Post Failed Final');

        eTestStep := E_BPTMTestStates.CleaningUp;
    END_IF

E_BPTMTestStates.CleaningUp:
    TEST_FINISHED_NAMED('BPTMErrorFullArb');

END_CASE

fbBPTM_TestFullArb(
    fbArbiter := fbArbFullErr,
    i_TransitionAssertionID := nTransitionID,
    i_stTransitionAssertion := stTransitionAssertion,

    i_nRequestedAssertionID := nReqID,
    i_stRequestedAssertion := stReqAssertion,

    stCurrentBeamParameters := fbSubSysIO.q_stSimulatedBPReadback,
);

fbSubSysIO(LA := fbArbFullErr, FFO := ffo);
END_METHOD

// Test the BPTM seamlessly handles new requests at any stage
// Verify old requests are removed from arbiter
{attribute 'no_check'}
METHOD InterruptAtAllSteps
VAR_INPUT
END_VAR
VAR
    //Final and transition assertions
    nTransitionID    :    UDINT := 16#DAAD;
    stTranReq    :    ST_BeamParams := PMPS_GVL.cst0RateBeam;

    nFirstReqID    :    UDINT    := 16#FEED;
    stFirstReq    :    ST_BeamParams := (nTran :=1, nRate := 16#FEED, neVRange :=2#1111_1111_1111_1111_1111_1111_1111_1111);

END_VAR
VAR_INST
    fbBPTM_InterruptionTest    :    BeamParameterTransitionManager;

    ffo : FB_HardwareFFOutput := (bAutoReset:=TRUE);
    fbSubSysIO : FB_DummyArbIO;
    fbBPR :  FB_BPRequestor;
    xFirstPass    :    BOOL := TRUE;
    eTestStep: E_BPTMTestStates := E_BPTMTestStates.Init;
    tonRetryTimeout : TON := (PT:=T#5s);

    fbBPTMDiscCycles : BeamParameterTransitionManager;
    fbSubSysIODisc : FB_DummyArbIO;
    fbArbDisc : FB_Arbiter(1000);

    iCount : UINT;

    aBPTM : ARRAY [1..cCycle] OF BeamParameterTransitionManager;
    BPTMUnderTest : REFERENCE TO BeamParameterTransitionManager;
    fbArbiter    :    FB_Arbiter(1);
    aArbIO : ARRAY [1..cCycle] OF FB_DummyArbIO;
    ArbIO : REFERENCE TO FB_DummyArbIO;
    nCycleLim : UINT;
    nCycle : UINT;
    sCurrentTestName : STRING :='';
    bCycleLimHit : BOOL;
    nAllStepsDone : BYTE;
    tTimeOut : TON := (PT:=T#20ms);

    bTestedOnce : BOOl;
END_VAR
VAR CONSTANT
    nNewTarget : INT := 0;
    nRequestBP : INT := 1;
    nWaitForBP : INT := 2;
    nTransitioning : INT := 3;
    nWaitForFinalBP : INT := 4;
    nCleaningUp : INT := 5;
    nDone : INT := 6;
    nIdle : INT := 7;
END_VAR

(* These tests will confirm the BPTM is interruptable at any step,
meaning it will not deadlock or stall, and will always complete with
the correct sequencing *)

(* This functionality is crucial as a deadlocked BPTM will need manual intervention,
users of the BPTM should always be able to just set a target BP that is easy to reach
at any point in time, and have the BPTM head in that direction and succeed. *)

// Determine how many cycles it would take normally, to complete a full BPTM cycle
// This count will be verified against the current count constant

IF NOT bTestedOnce THEN

TEST('CheckBPTM Cycle Count');

WHILE fbBPTMDiscCycles.eBPTMState <> E_BPTMState.Idle DO

    fbBPTMDiscCycles.i_TransitionAssertionID := nTransitionID;
    fbBPTMDiscCycles.i_stTransitionAssertion := stTranReq;

    fbBPTMDiscCycles.i_nRequestedAssertionID := nFirstReqID;
    fbBPTMDiscCycles.i_stRequestedAssertion := stFirstReq;

    fbBPTMDiscCycles(fbArbiter:=fbArbDisc);
    fbSubSysIODisc(LA:=fbArbDisc, FFO:=ffo);

    fbBPTMDiscCycles.stCurrentBeamParameters := fbSubSysIODisc.q_stSimulatedBPReadback;

    fbSubSysIODisc.AutoUpdateBP := TRUE;

    fbBPTMDiscCycles.i_xDoneMoving S= fbBPTMDiscCycles.q_xTransitionAuthorized;

    iCount := iCount + 1;
END_WHILE

IF fbBPTMDiscCycles.eBPTMState = E_BPTMState.Idle THEN
    AssertTrue(cCycle >= iCount, CONCAT('cCycle is too low, increase it to', INT_TO_STRING(iCount)));
    TEST_FINISHED_NAMED('CheckBPTM Cycle Count');
END_IF

// Run BPTM for nCycleLim cycles, switch to a new target, verify BPTM completes anyways

FOR nCycleLim := 1 TO cCycle DO

    nCycle := 0;

    bCycleLimHit := FALSE;

    BPTMUnderTest REF= aBPTM[nCycleLim];
    ArbIO REF= aArbIO[nCycleLim];

    BPTMUnderTest.i_TransitionAssertionID := nTransitionID;
    BPTMUnderTest.i_stTransitionAssertion := stTranReq;

    ArbIO.AutoUpdateBP := TRUE;

    // Start the test for this Cycle Limit
    sCurrentTestName := CONCAT('CycleLimTest:',INT_TO_STRING(nCycleLim));
    TEST(sCurrentTestName);

    nAllStepsDone := 0;

    tTimeOut(IN:=FALSE);

    WHILE nAllStepsDone <> 16#FF DO

        tTimeOut(IN:= TRUE);

        IF tTimeOut.Q THEN
            AssertTrue(FALSE, CONCAT('Failed ', BYTE_TO_HEXSTR(nAllStepsDone, 2, FALSE)));
            EXIT;
        END_IF

        // Verify all steps complete
        IF bCycleLimHit THEN
            nAllStepsDone.nNewTarget S= BPTMUnderTest.eBPTMState = E_BPTMState.NewTarget;
            nAllStepsDone.nRequestBP S= BPTMUnderTest.eBPTMState = E_BPTMState.RequestBP;
            nAllStepsDone.nWaitForBP S= BPTMUnderTest.eBPTMState = E_BPTMState.WaitForBP;
            nAllStepsDone.nTransitioning S= BPTMUnderTest.eBPTMState = E_BPTMState.Transitioning;
            nAllStepsDone.nWaitForFinalBP S= BPTMUnderTest.eBPTMState = E_BPTMState.WaitForFinalBP;
            nAllStepsDone.nCleaningUp S= BPTMUnderTest.eBPTMState = E_BPTMState.CleaningUp;
            nAllStepsDone.nDone S= BPTMUnderTest.eBPTMState = E_BPTMState.Done;
            nAllStepsDone.nIdle S= BPTMUnderTest.eBPTMState = E_BPTMState.Idle;
        ELSE
            nAllStepsDone := 0;
        END_IF

        // After nCycleLim cycles (nCycle), change the target
        IF nCycle >= nCycleLim THEN
            BPTMUnderTest.i_nRequestedAssertionID := nCycleLim;
            BPTMUnderTest.i_stRequestedAssertion.nRate := nCycleLim;
            bCycleLimHit := TRUE;
        ELSE
            BPTMUnderTest.i_nRequestedAssertionID := nFirstReqID;
            BPTMUnderTest.i_stRequestedAssertion := stFirstReq;
        END_IF

        BPTMUnderTest(fbArbiter:=fbArbiter);
        ArbIO(LA:=fbArbiter, FFO := ffo);

        BPTMUnderTest.stCurrentBeamParameters := ArbIO.q_stSimulatedBPReadback;

        BPTMUnderTest.i_xDoneMoving := BPTMUnderTest.q_xTransitionAuthorized;

        nCycle := nCycle + 1;

    END_WHILE

    AssertTrue(fbArbiter.CheckRequestInPool(BPTMUnderTest.i_nRequestedAssertionID),
        CONCAT('Final req not in pool: ', UINT_TO_STRING(nCycleLim)));
    AssertFalse(fbArbiter.CheckRequestInPool(BPTMUnderTest.i_TransitionAssertionID),
        'TransReq still in pool');
    AssertFalse(fbArbiter.CheckRequestInPool(nFirstReqID),
        'First req still in pool');
    AssertTrue(bCycleLimHit,
        CONCAT('Cycle lim not hit', UINT_TO_STRING(nCycleLim)));
    AssertTrue(ArbIO.q_stSimulatedBPReadback.nRate = BPTMUnderTest.i_stRequestedAssertion.nRate,
        'Rates are not equal...');

    TEST_FINISHED_NAMED(sCurrentTestName);

    // Clean up for next test

    fbArbiter.RemoveRequest(nFirstReqID);
    fbArbiter.RemoveRequest(nTransitionID);
    fbArbiter.RemoveRequest(nCycleLim);

END_FOR

END_IF
END_METHOD

// Test the BPTM seamlessly handles new requests at any stage
// Verify old requests are removed from arbiter
METHOD InterruptedTransition
VAR_INPUT
END_VAR
VAR
    //Final and transition assertions
    nTransitionID    :    UDINT := 3;
    stTranReq    :    ST_BeamParams := PMPS_GVL.cstSafeBeam;

    nFirstReqID    :    UDINT    := 1;
    stFirstReq    :    ST_BeamParams := (nRate := 100);

    nSecondReqID    :    UDINT    := 2;
    stSecReq    :    ST_BeamParams := (nRate:= 200);

END_VAR
VAR_INST
    fbBPTM_InterruptionTest    :    BeamParameterTransitionManager;
    fbArbiter    :    FB_Arbiter(1);
    ffo : FB_HardwareFFOutput;
    fbSubSysIO : FB_DummyArbIO;
    fbBPR :  FB_BPRequestor;
    xFirstPass    :    BOOL := TRUE;
    eTestStep: E_BPTMTestStates := E_BPTMTestStates.Init;
    tonRetryTimeout : TON := (PT:=T#5s);
END_VAR
CASE eTestStep OF

E_BPTMTestStates.Init:

    TEST('BPTM Intr Trans');

    fbBPTM_InterruptionTest.i_TransitionAssertionID := nTransitionID;
    fbBPTM_InterruptionTest.i_stTransitionAssertion := stTranReq;

    fbBPTM_InterruptionTest.i_nRequestedAssertionID := nFirstReqID;
    fbBPTM_InterruptionTest.i_stRequestedAssertion := stFirstReq;

    fbSubSysIO.AutoUpdateBP := TRUE; // Enable auto update

    eTestStep := E_BPTMTestStates.WaitingForTransitionAssertion;

E_BPTMTestStates.WaitingForBeam:

    IF fbBPTM_InterruptionTest.eBPTMState = E_BPTMState.WaitingForTransitionAssertion AND
        NOT fbBPTM_InterruptionTest.xEntry THEN // since we're not in entry anymore

        //change the request to interrupt
        fbBPTM_InterruptionTest.i_nRequestedAssertionID := nSecondReqID;
        fbBPTM_InterruptionTest.i_stRequestedAssertion := stSecReq;

        eTestStep := E_BPTMTestStates.Transitioning;
    END_IF

E_BPTMTestStates.Transitioning:

    TEST('New Target Gets To Trans Auth');

    tonRetryTimeout(IN:=TRUE);

    IF tonRetryTimeout.Q OR fbBPTM_InterruptionTest.q_xTransitionAuthorized THEN
        AssertTrue(fbBPTM_InterruptionTest.q_xTransitionAuthorized, 'Transition should have been authorized by now');
        AssertTrue(fbArbiter.CheckRequest(nTransitionID), 'Transition ID is missing from arbiter while transition is authorized');
        AssertTrue(fbArbiter.CheckRequest(nSecondReqID), 'Final ID is missing from arbiter while transition is authorized');

        TEST_FINISHED_NAMED('New Target Gets To Trans Auth');

        eTestStep := E_BPTMTestStates.CleaningUp;
    END_IF

E_BPTMTestStates.CleaningUp:
    TEST_FINISHED_NAMED('BPTM Intr Trans');

END_CASE

fbBPTM_InterruptionTest(
    fbArbiter := fbArbiter,
    stCurrentBeamParameters := fbSubSysIO.q_stSimulatedBPReadback
);

fbSubSysIO(LA := fbArbiter, FFO := ffo);
END_METHOD

END_FUNCTION_BLOCK

// ---- MajorComponents/BPTM/BeamParameterTransitionManager.TcPOU
(*
Implements the procedure for safely transitioning between device states.

NOTE:
The BPTM will throw an error if the arbiter does not have enough space for the transition and new final assertion.

 *)
{attribute 'no_check'}
FUNCTION_BLOCK BeamParameterTransitionManager
VAR_IN_OUT

    fbArbiter    :    FB_Arbiter; //Connect to local arbiter

END_VAR
VAR_INPUT
    i_sDeviceName	: 	STRING:='Device'; // Name of the device requesting the transition

    i_TransitionAssertionID    :    UDINT := 0; // Must not be 0 or EXCLUDED_ID
    i_stTransitionAssertion : ST_BeamParams := PMPS_GVL.cst0RateBeam; //Assertion required during transition (always safer than anything inbetween)

    i_nRequestedAssertionID    :    UDINT := 0; // Must not be 0 or EXCLUDED_ID
    i_stRequestedAssertion    :    ST_BeamParams := ( nTran := 0, neVRange := 0, nRate  := 0, nBCRange :=0);// PMPS_GVL.cstSafeBeam; //Requested assertion, change whenever

    i_xMoving    :    BOOL := FALSE; //Provide rising edge when device begins moving <remove>
    i_xDoneMoving    :    BOOL := FALSE; //Provide rising edge when device is done with a move

    stCurrentBeamParameters    :    ST_BeamParams := PMPS_GVL.cstFullBeam; //Connect to current beam parameters

    // Rising edge to cycle back through the BPTM process. Use if something in the process timed out or failed. This will interrupt a current process
    bRetry : BOOL := FALSE;
END_VAR
VAR_OUTPUT

    q_xTransitionAuthorized    :    BOOL := FALSE; //Rising edge indicating the device is safe to move, use as input to move execute (which requires a rising edge)

    bError : BOOL; // Set if some issue occurs within the bptm
    nErrId : UINT; // Set to non-zero to help understand the error.

    bDone : BOOL;
    bBusy : BOOL;

END_VAR

VAR
    nTargetAssertionID    :    UDINT := 0;
    stTargetAssertion    :    ST_BeamParams; // Target assertion
    nCurrentAssertionID    :    UDINT := 0;  // ID of last set state (zero until a state is reached)

    xNewBP    :    BOOL;
    xTranBP    :    BOOL;
    xFinalBPInArb : BOOL;
    xFinalBP    :    BOOL;

    eBPTMState : E_BPTMState := Init;
    ePrevState : E_BPTMState := Init;

    xEntry : BOOL;
    rTransition : R_TRIG;
    xNewTarget : BOOL;

    bTransAssertionFailed : BOOL;
    bFinalAssertionFailed : BOOL;

    LogStrBuffer : ARRAY [0..LogBuffSize] OF STRING;
    LogBuffIdx : FB_Index := (LowerLimit:=0, UpperLimit:=LogBuffSize);

    nAssrtAttempt : INT; // Number of times we have tried asserting a BP set

    rtRetry : R_TRIG;

    rtError : R_TRIG;

    ffTimeout : FB_FastFault := (
        i_Desc := 'Preemptive requests timed out in BPTM',
        i_TypeCode := 16#A,
        i_xAutoReset := FALSE);

    rtDoneMoving : R_TRIG;
    bLatchDoneMoving : BOOL;

    bFirstMove : BOOL := TRUE;

END_VAR
VAR CONSTANT
    LogBuffSize : INT := 40;
    cMaxAttempts : INT := 3;
    (* The thought here is, a BPTM needs at most 2 arbiter slots to complete a transition.
    If we're at capacity, it means some BPTM before this one has begun a transition,
    and will require at least one more arbiter spot to complete.
    *)
    cReqArbCapacity : UDINT := 2;
END_VAR


// Logic for retry button
rtRetry(CLK:=bRetry);
bRetry := FALSE;

// Logic for catching Move Done rising edge
rtDoneMoving(CLK:=i_xDoneMoving);
bLatchDoneMoving S= rtDoneMoving.Q;

// Logic for interrupting BPTM and changing requests
IF nTargetAssertionID <> i_nRequestedAssertionID OR rtRetry.Q THEN

    bError := FALSE;
    nErrID := 0;

    bDone := FALSE;
    bBusy := TRUE;

    // Execute exit actions before transition back to NewTarget
    CASE eBPTMState OF
        Transitioning:
            DeauthorizeTransition();
        //CleaningUp:
    END_CASE

    eBPTMState := E_BPTMState.NewTarget;
    xEntry := eBPTMState <> ePrevState;

END_IF

IF xEntry THEN nAssrtAttempt := 0; END_IF

rtError(CLK:=bError);

IF rtError.Q THEN
    eBPTMState := E_BPTMState.Error;
END_IF

// States
CASE eBPTMState OF
    NewTarget:
        IF xEntry THEN
            NewTarget_ENTRY();
        ELSIF xNewBP THEN
            eBPTMState := E_BPTMState.RequestBP;
        ELSE
            SetNewTarget();
        END_IF

    RequestBP:
        IF PMPS_PARAM.MAX_ASSERTIONS - fbArbiter.nEntryCount >= cReqArbCapacity THEN
            AssertTransitionBP();
            AssertFinalBP();
            eBPTMState := E_BPTMState.WaitForBP;
        ELSE
            LogActions('Arbiter at capacity, leaving space for other BPTM to finish.');
            nErrId := PMPS_CODES.NoRoomInArb;
            bError := TRUE;
        END_IF

    WaitForBP:
        WaitingForTransitionAssertion_DO();
        WaitingForFinalAssertion_DO();
        IF xTranBP AND xFinalBPInArb THEN eBPTMState := E_BPTMState.Transitioning; END_IF

    Transitioning:
        IF xEntry THEN
            AuthorizeTransition();
        ELSIF bLatchDoneMoving OR (bFirstMove AND i_xDoneMoving) THEN
            DeauthorizeTransition();
            eBPTMState := E_BPTMState.WaitForFinalBP;
        END_IF

    WaitForFinalBP:
        xFinalBP := F_SafeBPCompare(stCurrentBeamParameters, stTargetAssertion);
        IF xFinalBP THEN
            eBPTMState := E_BPTMState.CleaningUp;
        END_IF

    CleaningUp:
        IF xEntry THEN
            RemoveTransitionAssertion();
        ELSE
            eBPTMState := E_BPTMState.Done;
        END_IF

    Done:
        bDone := TRUE;
        bFirstMove := FALSE;
        LogActions('Returning to idle');
        eBPTMState := E_BPTMState.Idle;

    Error:
        bError := TRUE;
        eBPTMState := E_BPTMState.Idle;
END_CASE

xEntry := ePrevState <> eBPTMState;
ePrevState := eBPTMState;

bDone R= bError;
bBusy R= bError OR bDone;

ACTION AssertFinalBP:
//q_stFinalAssertion := stTargetAssertion;

//Clearing previous target parameters
(* This is considered safe at this step as the transition
state beam parameters should always be safer than the
current or target state beam parameters
*)
IF nCurrentAssertionID <> 0 THEN
    LogActions(CONCAT('Removing previous request: ', DWORD_TO_HEXSTR(nCurrentAssertionID, 4, false)) );
    fbArbiter.RemoveRequest( nCurrentAssertionID );
END_IF

LogActions(CONCAT('Asserting target req.: ', DWORD_TO_HEXSTR(nTargetAssertionID, 4, false)) );

//Asserting target parameters
bFinalAssertionFailed := NOT fbArbiter.AddRequest(
    nTargetAssertionID,
    stTargetAssertion,
    i_sDeviceName
);

IF bFinalAssertionFailed THEN
    LogActions('Assert final failed. ');
    nAssrtAttempt := nAssrtAttempt + 1;
    IF nAssrtAttempt > cMaxAttempts THEN
        bError := TRUE;
        nErrID := PMPS_CODES.FinalAssrtFail;
    END_IF
ELSE
    // Remembering final assertionID for removal later
    nCurrentAssertionID := nTargetAssertionID;
END_IF
END_ACTION

ACTION AssertTransitionBP:

LogActions( CONCAT('Removing transition id: ', DWORD_TO_STRING(i_TransitionAssertionID)) );
fbArbiter.RemoveRequest(i_TransitionAssertionID);

LogActions( CONCAT('Requesting transition id: ', DWORD_TO_STRING(i_TransitionAssertionID)) );
bTransAssertionFailed := NOT fbArbiter.AddRequest(
    i_TransitionAssertionID,
    i_stTransitionAssertion,
    i_sDeviceName
);

IF bTransAssertionFailed THEN
    LogActions('Assert trans. failed. ');
    nAssrtAttempt := nAssrtAttempt + 1;
    IF nAssrtAttempt > cMaxAttempts THEN
        bError := TRUE;
        nErrID := PMPS_CODES.TransAssrtFail;
    END_IF
END_IF
END_ACTION

ACTION AuthorizeTransition:
q_xTransitionAuthorized := TRUE;

bLatchDoneMoving R= q_xTransitionAuthorized;

LogActions('Authorizing transition');
END_ACTION

ACTION DeauthorizeTransition:
q_xTransitionAuthorized := FALSE;
LogActions('Deauthorizing transition');
END_ACTION

{attribute 'no_check'}
METHOD LogActions : BOOL
VAR_INPUT
    LogStr : STRING;
END_VAR
LogStrBuffer[LogBuffIdx.IncVal()] := LogStr;
END_METHOD

ACTION NewTarget_ENTRY:
xNewBP := False;
END_ACTION

ACTION RemoveTransitionAssertion:
//q_stTransitionAssertion := PMPS_GVL.cstFullBeam;

//Removing transition assertion
fbArbiter.RemoveRequest( i_TransitionAssertionID );

LogActions('Removing transition req');

//TODO add something to verify removal
END_ACTION

ACTION RequestBP_DO:
// Request BP atomically so we know we'll finish the BPTM cycle
IF fbArbiter.nEntryCount < cReqArbCapacity THEN

    LogActions( CONCAT('Removing transition id: ', DWORD_TO_STRING(i_TransitionAssertionID)) );
    fbArbiter.RemoveRequest(i_TransitionAssertionID);

    LogActions( CONCAT('Requesting transition id: ', DWORD_TO_STRING(i_TransitionAssertionID)) );
    bTransAssertionFailed := NOT fbArbiter.AddRequest(
        i_TransitionAssertionID,
        i_stTransitionAssertion,
        i_sDeviceName
    );

    IF bTransAssertionFailed THEN
        LogActions('Assert trans. failed. ');
        nAssrtAttempt := nAssrtAttempt + 1;
        IF nAssrtAttempt > cMaxAttempts THEN
            bError := TRUE;
            nErrID := PMPS_CODES.TransAssrtFail;
        END_IF
    END_IF



ELSE
    LogActions('Arbiter at capacity, leaving space for other BPTM to finish.');
END_IF
END_ACTION

ACTION SetNewTarget:

IF F_ValidReqID(i_nRequestedAssertionID) AND
    F_ValidReqID(i_TransitionAssertionID) THEN

    stTargetAssertion := i_stRequestedAssertion;
    nTargetAssertionID := i_nRequestedAssertionID;

    LogActions('New target set');

    xNewBP := TRUE;

ELSE
    IF NOT F_ValidReqID(i_nRequestedAssertionID) THEN

        nErrID := PMPS_CODES.BadTargetID;
    ELSIF NOT F_ValidReqID(i_TransitionAssertionID) THEN
        nErrID := PMPS_CODES.BadTransID;
    END_IF
    LogActions('Error in set new target');
    bError := TRUE;
END_IF
END_ACTION

ACTION WaitingForFinalAssertion_DO:
//Final Assertion Verification

xFinalBPInArb := fbArbiter.CheckRequest( i_nRequestedAssertionID);;
END_ACTION

ACTION WaitingForFinalAssertion_EXIT:
//Set this bool false so we can get a rising edge on the next try
xFinalBP := FALSE;
END_ACTION

ACTION WaitingForTransitionAssertion_DO:
//Transition Assertion Verification
xTranBP    := F_SafeBPCompare0Rate(stCurrentBeamParameters, i_stTransitionAssertion) AND
    fbArbiter.CheckRequest(i_TransitionAssertionID);
END_ACTION

ACTION WaitingForTransitionAssertion_EXIT:
xTranBP := FALSE;
END_ACTION

END_FUNCTION_BLOCK

// ---- MajorComponents/Arbiter/FB_Arbiter.TcPOU
(* FB Arbiter
A. Wallace 2020-6-26

The arbiter primary objectives are:
- Provide a simple interface for devices to request beam parameter sets
- Provide a way for devices to verify their BPS is active in the arbiter
- Provide a way for devices remove their requests from evaluation
- Evaluate all active beam parameter requests registered with the aribiter,
to determine the safest combination of all sets, provide this set as an output.
- Do all of this with minimal overhead

To these ends, the arbiter uses a hash-table, the rows being a state-id as the key, and a corresponding
 beam parameter set to be evaluated against all the other sets (or rows), in the table.

The hash table can be thought of as an array on steriods, they are worth reading about, suffice to say
the hash table will tell you when you reach the end of all the entries, and enables us to find entries quickly.

These features efficiently address the addition, removal, and verification of beam parameter sets listed in the above requirements.
*)
{attribute 'reflection'}
FUNCTION_BLOCK FB_Arbiter IMPLEMENTS I_HigherAuthority, I_LowerAuthority
VAR
    nRequestsCount : UDINT; // How many requests are currently in the arbiter

    {attribute 'pytmc' := '
        pv: AP
        io: i
        field: DESC Assertion Pool
     '}
    fbBPAssertionPool    :    FB_BeamParamAssertionPool; //Table of active beam parameter assertions

    xRequestMade : BOOL; // Arbiter has confirmed its request has made it into the beam parameter request

    {attribute 'pytmc' := '
        pv: ArbiterID
        io: i
        field: DESC Arbiter ID for elev. req.
     '}
    nArbiterID : UDINT; // Arbiter ID, used for making higher-level BP requests

    nNextCohort : UDINT := 1; // The cohort ID any new requests will adopt, will become ReqInProgCohort at the start of the next acknowledgement cycle
    nAckInProgCohort : UDINT := 0; // The cohort ID currently being acknowledged, will become nActiveCohort after acknowledgement from HA
    {attribute 'pytmc' := '
        pv: CohortCounter
        io: i
        field: DESC Intrnl cohort counter
     '}
    nActiveCohort : UDINT := 0; // Requests with cohorts <= to this value will be considered active in CheckRequest

    bStartNewAckRequest : BOOL; // Set by an add or remove method call, triggers an ack cycle
    bAckInProgress : BOOL; // Set by ElevateReq when there is a new ack request and reset when the ack cycle is complete

    // The following IDs are set by the last BP request that was most conservative
    // ie. other requests may limit the parameter, but this one is the most recent to limit it
    idTransmission : DWORD; // ID of BP limiting transmission
    idRate : DWORD; // ID of BP limiting rate

    {attribute 'instance-path'}
    {attribute 'noinit'}
    sPath    :    T_MaxString;

    sArbName : T_MaxString;

    InfoStringFmtr : FB_FormatString;

    bVerbose : BOOL := FALSE;

    {attribute 'pytmc' := '
        pv: Vetoed
        io: i
        field: DESC Arbiter Veto Status
    '}
    bArbiterVetoed : BOOL := FALSE;
END_VAR
VAR_INPUT
END_VAR
VAR_OUTPUT
    {attribute 'pytmc' := '
        pv: ArbitratedBP
        io: i
        field: DESC Arbitrated BP
     '}
    q_stBeamParams    :    ST_BeamParams := PMPS_GVL.cstFullBeam; //Updated on each cycle of the arbiter FB with the current arbitrated beam parameter set

    q_xStateIDFound    :    BOOL; //Set true if a state-id is found in the assertion pool after calling A_VerifyAssertion
END_VAR

// Adds a request to the arbiter pool.
// Returns true if the request was successfully added, false if not enough space or a request with the same ID is already present.
METHOD AddRequest : BOOL
VAR_INPUT
    nReqID    :    DWORD; // Unique ID within aribter for the request. Make sure this is unique for every device + state combination
    stReqBP        :    ST_BeamParams; //Requested beam params
    sDevName: STRING; // Name of the device making the request
END_VAR
VAR
    BP_Int : ST_BP_ArbInternal;
END_VAR
VAR_INST
    fbLog : FB_LogMessage;
END_VAR
// If the request is already in the pool, then skip the rest.
// This is flawed, needs to update the request if it's already in the pool, despite having the same ID
IF THIS^.CheckRequestInPool(nReqID)
    OR nReqID = PMPS_GVL.EXCLUDED_ASSERTION_ID
    OR nReqID = 0 THEN
    AddRequest := FALSE;
    RETURN;
END_IF


stReqBP.nCohortInt := nNextCohort; // Set the cohort number for this BP request.

// Pack the ID with the request
MEMCPY(ADR(BP_Int), ADR(stReqBP), SIZEOF(stReqBP));
BP_Int.nId := nReqID;
BP_Int.LiveInTable := TRUE;
BP_Int.sDevName := sDevName;

THIS^.fbBPAssertionPool.A_Add(
    key := nReqID,
    putValue := BP_Int
);


IF NOT THIS^.fbBPAssertionPool.bOk THEN
    fbLog(sMsg:=CONCAT('Addition to arbiter assertion pool failed ', DWORD_TO_HEXSTR(nReqID, 4, FALSE)),
            eSevr:=TcEventSeverity.Warning,
            eSubsystem:=E_Subsystem.MPS,
            sJson := F_PMPS_JSON(
                        sArbName,
                        sPath,
                        PMPS_CODES.ARB_FULL));
ELSIF THIS^.fbBPAssertionPool.bOk AND bVerbose THEN
    fbLog(sMsg:=CONCAT('Added to pool ',DWORD_TO_HEXSTR(nReqID, 4, FALSE)),
            eSevr:=TcEventSeverity.Verbose,
            eSubsystem:=E_Subsystem.MPS);
END_IF
// New request, make sure the ack cycle request flag is set
bStartNewAckRequest S= THIS^.fbBPAssertionPool.bOk;

AddRequest := THIS^.fbBPAssertionPool.bOk;

nRequestsCount := nEntryCount;
END_METHOD

// Kernel of the arbiter
// Logic for determining which beam parameter is the most conservative across all request sets.
{attribute 'no_check'}
METHOD INTERNAL ArbitrateBP : ST_BP_ArbInternal
VAR_INPUT
    stBP1    :    ST_BP_ArbInternal;
    stBP2    :    ST_BP_ArbInternal;
END_VAR
VAR
    idx : UINT := 1;
    bcBitmask : WORD:=0;
END_VAR
//<TODO>Add something here to register the key that won for each param

//Attenuation
ArbitrateBP.nTran := MIN(stBP1.nTran, stBP2.nTran);

FOR idx := 1 TO PMPS_GVL.AUX_ATTENUATORS DO
    ArbitrateBP.astAttenuators[idx].nTran := MIN(stBP1.astAttenuators[idx].nTran, stBP2.astAttenuators[idx].nTran);
END_FOR

//Apertures
FOR idx := 1 TO PMPS_GVL.MAX_APERTURES DO
    IF stBP1.astApertures[idx].Height = 0 OR stBP2.astApertures[idx].Height =0 THEN
        ArbitrateBP.astApertures[idx].Height := MAX(stBP1.astApertures[idx].Height, stBP2.astApertures[idx].Height);
    ELSE
        ArbitrateBP.astApertures[idx].Height := MIN(stBP1.astApertures[idx].Height, stBP2.astApertures[idx].Height);
    END_IF

    IF stBP1.astApertures[idx].Width = 0 OR stBP2.astApertures[idx].Width =0 THEN
        ArbitrateBP.astApertures[idx].Width := MAX(stBP1.astApertures[idx].Width, stBP2.astApertures[idx].Width);
    ELSE
        ArbitrateBP.astApertures[idx].Width := MIN(stBP1.astApertures[idx].Width, stBP2.astApertures[idx].Width);
    END_IF
END_FOR

//Photon energy ranges
ArbitrateBP.neVRange := stBP1.neVRange AND stBP2.neVRange;

//Beam Class ranges
ArbitrateBP.nBCRange := stBP1.nBCRange AND stBP2.nBCRange;

//Beam Class
//Assert the highest allowed beamclass
IF (ArbitrateBP.nBCRange = 0) THEN ArbitrateBP.nBeamClass := 0; END_IF
FOR idx:=1 TO 15 BY 1 DO
    IF (idx =1 ) THEN bcBitmask :=1; END_IF
    IF (ArbitrateBP.nBCRange AND bcBitmask) = bcBitmask THEN
        ArbitrateBP.nBeamClass := TO_USINT(idx);
    END_IF
    bcBitmask := ROL(bcBitmask,1);
END_FOR


//Rate
ArbitrateBP.nRate := MIN(stBP1.nRate, stBP2.nRate);
END_METHOD

PROPERTY bLowerAuthorityVetoed : BOOL
GET
bLowerAuthorityVetoed := bArbiterVetoed;
END_GET
SET
bArbiterVetoed := bLowerAuthorityVetoed;
END_SET
END_PROPERTY

(* Checks request ID is included in arbitration all the way to the accelerator interface
Use like so:
IF fbArbiter.CheckRequest(nStateIDAssertionToCheck) AND (other logic) THEN:
    Request is found and active in arbitration,. Do something.
ELSE:
    Request was not found, or is not yet included in arbitration. Don't do something/ wait.

*)
METHOD CheckRequest : BOOL
VAR_INPUT
    nReqID    :    DWORD;
END_VAR
VAR
    BP : ST_BeamParams;
END_VAR
fbBPAssertionPool.A_Lookup(key := nReqID);

// Verify BP is acknowledged
BP := fbBPAssertionPool.getValue;

// This logic:
// Did we find the assertion in the pool?
// Is the assertion cohort number less than the current cohort and greater than zero?
// Is the Aribter itself active in arbitration?
CheckRequest := fbBPAssertionPool.bOk AND
                BP.nCohortInt <= nActiveCohort AND
                BP.nCohortInt > 0;
END_METHOD

// Verify request is at least in the local arbiter
// Does not verify request has been included in arbitration.
// Use CheckRequest instead.
METHOD CheckRequestInPool : BOOL
VAR_INPUT
    nReqID    :    DWORD;
END_VAR
THIS^.fbBPAssertionPool.A_Lookup(key := nReqID);

CheckRequestInPool := THIS^.fbBPAssertionPool.bOk;
END_METHOD

// <Arbiter Internal>
// Elevates the arbitrated BP set to something above.
// Could be another arbiter, or a BP requester/ IO,
// or an FB that locks in a specific portion of the BP set.
METHOD ElevateRequest : BOOL
VAR_INPUT
    HigherAuthority : I_HigherAuthority;
END_VAR
(*
This method should only be used with one higher level component.
*)

// Complete previous ack cycle
IF bAckInProgress THEN
    IF HigherAuthority.CheckRequest(nReqID := nArbiterID) THEN
        nActiveCohort := nAckInProgCohort;
        bAckInProgress := FALSE;
    END_IF
END_IF

// Kick off another ack cycle
IF bStartNewAckRequest AND NOT bAckInProgress THEN
    nAckInProgCohort := nNextCohort;
    HigherAuthority.RemoveRequest(nReqID:= nArbiterID);
    bAckInProgress := HigherAuthority.RequestBP(nReqID := nArbiterID, stReqBP := GetArbitratedBP());
    IF bAckInProgress THEN
        bStartNewAckRequest := FALSE;
        nNextCohort := nNextCohort + 1;
    END_IF
END_IF
END_METHOD

METHOD FB_init : BOOL
VAR_INPUT
    bInitRetains : BOOL; // if TRUE, the retain variables are initialized (warm start / cold start)
    bInCopyCode : BOOL;  // if TRUE, the instance afterwards gets moved into the copy code (online change)
    nID : DWORD := PMPS_GVL.EXCLUDED_ASSERTION_ID; // Arbiter ID, must be globally unique cannot be zero or 16#FFFF
END_VAR
nArbiterID := nId;
fbBPAssertionPool.A_Reset();

sArbName := CONCAT('Arbiter ID: 0x', DWORD_TO_HEXSTR(nID, 4, FALSE));
END_METHOD

// Executes Arbitration between all requested beam parameter sets
METHOD INTERNAL GetArbitratedBP : ST_BeamParams
VAR_INPUT
END_VAR
VAR
    getPosPtr    : POINTER TO T_HashTableEntry := 0;
    getBPStructInt    :    ST_BP_ArbInternal;
    stOutputBP    :    ST_BP_ArbInternal; //Holding struct for arbitration process
END_VAR
VAR_INST
    xFirstPass : BOOL := TRUE;
    fbGetCurTaskIdx : GETCURTASKINDEX;
    LastCycleCount : UDINT;
    fbLogMessage : FB_LogMessage;
END_VAR
//Arbitrate
(*
This step cycles through every hash table entry, comparing
the beam parameters from each assertion to what we're planning
to assert.

The safer of the two parameters is kept so at the end we may
have a mix of beam parameters, the composition being safe for
all asserters.

*)

THIS^.fbBPAssertionPool.A_GetFirst( putPosPtr := 0, getPosPtr=>getPosPtr, getValue=>getBPStructInt );
IF THIS^.fbBPAssertionPool.bOk THEN //If the table is empty (not OK), we are left with the default stOutputBP set above.

    //The first entry in the hash table is taken as the setting to arbitrate against
    stOutputBP := getBPStructInt;

    REPEAT
        THIS^.fbBPAssertionPool.A_GetNext( putPosPtr := THIS^.fbBPAssertionPool.getPosPtr, getPosPtr=>getPosPtr, getValue=>getBPStructInt );
        IF THIS^.fbBPAssertionPool.bOk THEN
            stOutputBP := ArbitrateBP(stOutputBP, getBPStructInt);
        END_IF
    UNTIL NOT fbBPAssertionPool.bOk
    END_REPEAT
ELSE
    //Full beam if there are no arbitration requests
    MEMCPY(ADR(stOutputBP), ADR(PMPS_GVL.cstFullBeam), SIZEOF(PMPS_GVL.cstFullBeam));
END_IF

MEMCPY(ADR(q_stBeamParams),ADR(stOutputBP), SIZEOF(q_stBeamParams));

GetArbitratedBP := stOutputBP;

GetArbitratedBP.xValidToggle := NOT GetArbitratedBP.xValidToggle;

xFirstPass := FALSE;
END_METHOD

// How many entries are in the arbiter now
PROPERTY nEntryCount : UDINT
GET
fbBPAssertionPool.A_Count();
IF fbBPAssertionPool.bOk THEN
    nEntryCount := fbBPAssertionPool.nCount ;
END_IF
END_GET
END_PROPERTY

PROPERTY nLowerAuthorityID : DWORD
GET
nLowerAuthorityID := nArbiterID;
END_GET
END_PROPERTY

(* Removes request from abritration. *)
METHOD RemoveRequest : BOOL
VAR_INPUT
    nReqId    :    DWORD;
END_VAR
VAR_INST
    fbLog : FB_LogMessage;
END_VAR
VAR CONSTANT
    BP_Int : ST_BP_ArbInternal := (nId:=0, LiveInTable:=FALSE);
END_VAR
IF nReqId <> PMPS_GVL.EXCLUDED_ASSERTION_ID AND CheckRequestInPool(nReqId) THEN
    // Include an A_Add action here to
    // update this entry with a dummy filler (ID = 0, LiveInTable= False)
    // before removing it since this hash
    // table needs to be viewed with a diagnostic
    // and so the entries need to appear clean.
    THIS^.fbBPAssertionPool.A_Add(key := nReqID, putValue := BP_Int);
    THIS^.fbBPAssertionPool.A_Remove(key := nReqId);

    IF bVerbose THEN
        IF THIS^.fbBPAssertionPool.bOk THEN
                fbLog(sMsg:=CONCAT('Removed from pool: ', DWORD_TO_HEXSTR(nReqID,4,FALSE)),
                eSevr:=TcEventSeverity.Verbose,
                eSubsystem:=E_Subsystem.MPS);
        ELSE
            fbLog(sMsg:=CONCAT('Failed to remove from pool: ', DWORD_TO_HEXSTR(nReqID,4,FALSE)),
                eSevr:=TcEventSeverity.Warning,
                eSubsystem:=E_Subsystem.MPS);
        END_IF
    END_IF

    // With any new request reset the internal arbiter "done" flag
    bStartNewAckRequest S= THIS^.fbBPAssertionPool.bOk;

    RemoveRequest := THIS^.fbBPAssertionPool.bOk;

    nRequestsCount := nEntryCount;

END_IF
END_METHOD

METHOD RequestBP : BOOL
VAR_INPUT
    (*StateID of state requesting beam parameter set*)
    nReqID	: DWORD;
    (*Requested beam params*)
    stReqBP	: ST_BeamParams;
END_VAR
RequestBP := AddRequest(nReqID := nReqID, stReqBP := stReqBP, sDevName:=sArbName);
END_METHOD

END_FUNCTION_BLOCK

// ---- MajorComponents/Arbiter/FB_BeamParamAssertionPool.TcPOU
(* This function block implements simple database. Data element values are stored in the hash table.  *)
{attribute 'no_check'}
FUNCTION_BLOCK FB_BeamParamAssertionPool
VAR_INPUT
    key         : DWORD := 0;(* Entry key: used by A_Lookup, A_Remove method, the key variable is also used by A_Add method *)
    putPosPtr    : POINTER TO T_HashTableEntry := 0;(* Hash table entry position pointer (used by A_Find, A_GetNext, A_GetPrev) *)
    putValue     : ST_BP_ArbInternal;(* Hash table entry value (used by A_AddHead, A_AddTail, A_Find )*)
END_VAR
VAR_OUTPUT
    bOk            : BOOL := FALSE;(* TRUE = Success, FALSE = Failed *)
    getPosPtr    : POINTER TO T_HashTableEntry := 0;(* Returned hash table entry position pointer *)
    getValue     : ST_BP_ArbInternal;(* Returned hash table entry value *)
    nCount        : UDINT := 0;(* Hash table size (number of used entries, used by A_Count) *)
END_VAR
VAR
    {attribute 'pytmc' := '
        pv: Entry
        io: i
     '}
    epicsDataPool    : ARRAY[1..PMPS_PARAM.MAX_ASSERTIONS] OF ST_BP_ArbInternal;(* Structured data element pool for display in EPICS*)
    dataPool    : ARRAY[0..PMPS_PARAM.MAX_ASSERTIONS*3] OF ST_BP_ArbInternal;(* Structured data element pool *)
    entries        : ARRAY[0..PMPS_PARAM.MAX_ASSERTIONS*3] OF T_HashTableEntry;(* Max. number of hash table entries. The value of table entry = 32 bit integer (pointer to dataPool-array-entry) *)
    fbTable     : FB_HashTableCtrl;(* basic hash table control function block *)
    hTable         : T_HHASHTABLE;(* hash table handle *)
    pRefPtr        : POINTER TO ST_BP_ArbInternal := 0;
    indexOfElem    : ULINT;(* Integer value (max. size: x86=>32bit, x64=>64bit)*)
    cstSafeBeam :ST_BeamParams := ( nTran := 0, neVRange := 0, nRate  := 0, nBCRange :=0);// MG
END_VAR

;

ACTION A_Add:
(* Adds entry to the table *)
MEMSET( ADR( getValue ), 0, SIZEOF( getValue ) );
getPosPtr := 0;

fbTable.A_Add( hTable := hTable, key := key, putValue := ADR(cstSafeBeam)(* we will set this value later *), getPosPtr=>getPosPtr, bOk=>bOk );(* Add new element to the table, getPosPtr points to the new entry *)
IF fbTable.bOk THEN(* Success *)
    fbTable.A_GetIndexAtPosPtr( hTable := hTable, putPosPtr := getPosPtr, getValue =>indexOfElem, bOk=>bOk );(* Get array index of getPosPtr entry *)
    IF fbTable.bOk THEN(* Success *)
        pRefPtr     := ADR( dataPool[indexOfElem] );(* Get pointer to the data element *)

        pRefPtr^ := putValue;(* copy application value *)

        fbTable.A_Add( hTable := hTable, key := key, putValue := pRefPtr, bOk=>bOk );(* Assign the entry value = pointer to the data element *)
        IF fbTable.bOk THEN(* Success *)
            getValue := putValue;
        END_IF
    END_IF
END_IF

DataPoolToEpics();
END_ACTION

ACTION A_Count:
(* Count number of used entries *)
nCount := hTable.nCount;
bOk := TRUE;
END_ACTION

ACTION A_GetFirst:
(* Get first entry position pointer and value *)
MEMSET( ADR( getValue ), 0, SIZEOF( getValue ) );
getPosPtr := 0;

fbTable.A_GetFirst( hTable := hTable, putPosPtr := putPosPtr, getValue=>pRefPtr, getPosPtr=>getPosPtr, bOk=>bOk );
IF fbTable.bOk THEN
    getValue := pRefPtr^;
END_IF
END_ACTION

ACTION A_GetNext:
(* Get next entry position pointer and value *)
MEMSET( ADR( getValue ), 0, SIZEOF( getValue ) );
getPosPtr := 0;
bOk := FALSE;

IF putPosPtr = 0 THEN
    RETURN;
END_IF

fbTable.A_GetNext( hTable := hTable, putPosPtr := putPosPtr, getValue=>pRefPtr, getPosPtr=>getPosPtr, bOk=>bOk );
IF fbTable.bOk THEN
    getValue := pRefPtr^;
END_IF
END_ACTION

ACTION A_Lookup:
(* Lookup for entry by key  *)
MEMSET( ADR( getValue ), 0, SIZEOF( getValue ) );
getPosPtr := 0;

fbTable.A_Lookup( key := key, hTable := hTable, putPosPtr := putPosPtr, getValue=>pRefPtr, getPosPtr=>getPosPtr, bOk=>bOk );
IF fbTable.bOk THEN
    getValue := pRefPtr^;
END_IF
END_ACTION

ACTION A_Remove:
(* Search for entry and remove it *)
MEMSET( ADR( getValue ), 0, SIZEOF( getValue ) );
getPosPtr := 0;

fbTable.A_Remove( key := key, hTable := hTable, putPosPtr := putPosPtr, getValue=>pRefPtr, getPosPtr=>getPosPtr, bOk=>bOk );
IF fbTable.bOk THEN
    getValue := pRefPtr^;
END_IF

DataPoolToEpics();
END_ACTION

ACTION A_Reset:
(* Reset/initialize linked list *)
MEMSET( ADR( getValue ), 0, SIZEOF( getValue ) );
getPosPtr := 0;
bOk := F_CreateHashTableHnd( ADR( entries ), SIZEOF( entries ), hTable );(* Intialize table handle *)
fbTable.A_Reset( hTable := hTable, bOk=>bOk );
nCount := 0;
END_ACTION

ACTION DataPoolToEpics:

MEMCPY(ADR(epicsDataPool), ADR(dataPool), (PMPS_PARAM.MAX_ASSERTIONS) * SIZEOF(ST_BP_ArbInternal));
END_ACTION

END_FUNCTION_BLOCK

// ---- HelperFunctions/F_PMPS_JSON.TcPOU
FUNCTION F_PMPS_JSON : STRING
VAR_INPUT
    sDevName : STRING := '';
    sPath : STRING := '';
    nTypeCode : UINT := 0;
END_VAR
VAR

END_VAR


PMPS_TOOLS.fbJson.StartObject();
PMPS_TOOLS.fbJson.AddKey('pmps_typecode');
PMPS_TOOLS.fbJson.AddUdint(nTypeCode);
PMPS_TOOLS.fbJson.AddKey('pmps_path');
PMPS_TOOLS.fbJson.AddString(sPath);
PMPS_TOOLS.fbJson.AddKey('pmps_device_name');
PMPS_TOOLS.fbJson.AddString(sDevName);
PMPS_TOOLS.fbJson.EndObject();
F_PMPS_JSON := PMPS_TOOLS.fbJson.GetDocument();
PMPS_TOOLS.fbJson.ResetDocument();

END_FUNCTION

// ---- MajorComponents/FastFaults/FB_FastFault.TcPOU
(* Fast Fault
2019-9-13 A. Wallace

Use this block to generate a beam-off fault. Connects to a fast fault hardware output
function block to contribute to the state of the fast fault output (FFO).

If the i_xOK goes false, the associated FFO will go false, despite the state of any other
contributing fast faults, unless the FFO is currently vetoed.

*)
{attribute 'reflection'}
FUNCTION_BLOCK FB_FastFault
VAR_INPUT

    i_xOK        :    BOOL; // Connect to fast-fault condition (false produces fault)
    i_xReset    :    BOOL; // Resets when i_xOK is true and this is true
    i_xAutoReset : BOOL := FALSE; // Automatically clear fast fault (latching vs non-latching)
    i_xVetoable : BOOL := TRUE; // Mask this fast fault if the FFO veto device is true

    i_DevName : T_MaxString := ''; // Device name for diagnostic
    i_Desc : T_MaxString := ''; // Description of fast fault (you should set at init)
    i_TypeCode : UINT; // Error code for classifying fast faults
END_VAR
VAR_OUTPUT
    o_xFFLine    :    BOOL; //Connect to HW output or another FF input if you like (Optional)
END_VAR
VAR_IN_OUT
    io_fbFFHWO        :    FB_HardwareFFOutput; //Point to FB_HardwareFFOutput of your choice
END_VAR
VAR
    {attribute 'instance-path'}
    {attribute 'noinit'}
    sPath    :    T_MaxString;

    FFInfo : ST_FFInfo;

    RegistrationIdx : UINT := 1; // The index this FF was registered in the FFO

    xInit    :    BOOL :=TRUE;

    InfoStringFmtr : FB_FormatString;

    InUse : T_MaxString;
    AutoReset : T_MaxString;

END_VAR

IF xInit    THEN
    FFInfo.sPath := sPath;
    FFInfo.InUse := True;
    FFInfo.TypeCode := i_TypeCode;
    FFInfo.DevName := i_DevName;
    FFInfo.Desc := i_Desc;
    FFInfo.AutoReset := i_xAutoReset;
    FFInfo.Vetoable := i_xVetoable;

    InUse := BOOL_TO_STRING(FFInfo.InUse);
    AutoReset := BOOL_TO_STRING(FFInfo.AutoReset);
    InfoStringFmtr(sFormat:='%s;%s;%X;%s;%s;%s;',
        arg1 := F_STRING(FFinfo.sPath),
        arg2 := F_STRING(InUse),
        arg3 := F_WORD(FFInfo.TypeCode),
        arg4 := F_STRING(FFInfo.DevName),
        arg5 := F_STRING(FFInfo.Desc),
        arg6 := F_STRING(AutoReset),
        sOut=>FFInfo.InfoString);
    io_fbFFHWO.Register(
        stFFInfo:=FFInfo,
        Idx=>RegistrationIdx);
    //<TODO> if registration doesn't succeed, send warning to diagnostic
    xInit := FALSE;
END_IF

io_fbFFHWO.IdxCheckIn(Idx:=RegistrationIdx, OK := i_xOK, Reset:= i_xReset);

END_FUNCTION_BLOCK

// ---- MajorComponents/FastFaults/FB_HardwareFFOutput.TcPOU
{attribute 'reflection'}
{attribute 'no_check'}
FUNCTION_BLOCK FB_HardwareFFOutput EXTENDS FB_StopperVetoable
VAR CONSTANT
    FF_ARRAY_UPPER_BOUND : UINT := PMPS_PARAM.MAX_FAST_FAULTS;
END_VAR
VAR_INPUT
    {attribute 'pytmc' := '
        pv: ClearFault
        io: o
        field: DESC Might be overidden by PLC writes
     '}
    i_xReset    :    BOOL;
    {attribute 'pytmc' := '
        pv: EnableVeto
        io: o
     '}
    i_xVeto    :    BOOL;
    bAutoReset : BOOL := FALSE; // Set true for the FFO to automatically permit beam again after all fast faults are cleared
    i_sNetID : T_AmsNetID:=''; //Set to the Arbiter AmsNetID to be used for the synchronisation. An empty string means the system will sue local time
END_VAR
VAR_OUTPUT
    {attribute 'pytmc' := '
        pv: FaultHWO
        io: i
        field: DESC Hardware Output Status
     '}
    q_xFastFaultOut    AT %Q*    :    BOOL;
    q_xValidSyncTime : BOOL;// system time bValid output True when sync is successful
END_VAR
VAR_IN_OUT

END_VAR
VAR
    {attribute 'pytmc' := '
        pv: FF
     '}
    astFF : ARRAY[1..FF_ARRAY_UPPER_BOUND] OF ST_FF;

    {attribute 'pytmc' := '
        pv: RegistrationFailure
        io: io
     '}
    xFastFaultRegFail  :   BOOL := FALSE; // Set true if a fast fault fails to register. Holds beam off.
    tFFRegFail : F_TRIG;

    {attribute 'instance-path'}
    {attribute 'noinit'}
    sPath    :    T_MaxString;

    {attribute 'pytmc' := '
        pv: OK
        io: i
     '}
    xOK    :    BOOL:= TRUE; // Current internal state of FFO, indicates if FFO will accept a reset

    rtReset    :    R_TRIG;
    rtResetandOK : R_TRIG;

    nIndex    :    UINT := 1;

    IdxOK: BOOL;

    fbTime : FB_LocalSystemTime := ( bEnable := TRUE, dwCycle := 1 ); //Get current system time, used for override
    fbTime_to_UTC: FB_TzSpecificLocalTimeToSystemTime;
    fbGetTimeZone: FB_GetTimeZoneInformation;
    fbJson : FB_JsonSaxWriter;
    pmpsTypeCode : UDINT := 0; // shows up in json as pmps_typecode
    fbLogger : FB_LogMessage := (
        eSevr := TcEventSeverity.Critical,
        eSubsystem := E_Subsystem.MPS,
        nMinTimeViolationAcceptable := PMPS_PARAM.MAX_FAST_FAULTS);

END_VAR

// <TODO> latch off beam if DI card status goes bad

ACTION EvaluateOutput:

////////////////////////////////////////////////////////////////
// Critical code. Do not touch unless you know what you're doing
////////////////////////////////////////////////////////////////

//<TODO> add diagnostic for success or failure of reset
rtReset(CLK:=i_xReset);
rtResetandOK(CLK:=(rtReset.Q OR bAutoReset) AND xOK);

q_xFastFaultOut S= rtResetandOK.Q;
q_xFastFaultOut R= (NOT xOK OR xFastFaultRegFail);

//Reset OK for next cycle
xOK := True;

////////////////////////////////////////////////////////////////
END_ACTION

{attribute 'no_check'}
METHOD EvaluateOverrides : BOOL
VAR_INPUT
END_VAR
VAR
    FF : REFERENCE TO ST_FF;
    EvalIdx: DINT := 1;
END_VAR
VAR CONSTANT
    MaxTime : DINT:= 4294080;(*49.7 days*)
END_VAR
//Get local System Time
fbTime(sNetID:=i_sNetID);
//Get Time Zone
fbGetTimeZone(sNetID:=i_sNetID,bExecute:=TRUE,tTimeout:=T#10S);
//change local time to UTC to be compatible with unix time epoch widget
fbTime_to_UTC(in:= fbTime.systemTime , tzInfo:=fbGetTimeZone.tzInfo);
q_xValidSyncTime := fbTime.bValid AND NOT fbGetTimeZone.bError;

FOR EvalIdx := 1 TO FF_ARRAY_UPPER_BOUND DO

    FF REF= astFF[EvalIdx];

    IF NOT FF.Info.InUse THEN
        CONTINUE;
    ELSE
        // Veto timer
        IF FF.Ovrd.Deactivate THEN
            FF.Ovrd.Timer.PT := T#0s; // Only needs to be set zero for one cycle
        ELSIF FF.Ovrd.Activate THEN
            FF.Ovrd.StartDT:= TO_DINT(TO_DT(SystemTime_TO_DT(fbTime_to_UTC.out)));
            IF (FF.Ovrd.StartDT < FF.Ovrd.Expiration) THEN
                FF.Ovrd.Expiration:= LIMIT(0,FF.Ovrd.Expiration, FF.Ovrd.StartDT+MaxTime );
                   FF.Ovrd.Timer.PT := TO_DT(FF.Ovrd.Expiration)- SystemTime_TO_DT(fbTime_to_UTC.out);
            END_IF
        END_IF

        // UDINT conversions for ESS module compatibility.
        FF.Ovrd.Timer(
            IN := FF.Ovrd.Activate, // Rising edge activated
            Q => FF.Ovrd.Active);

        FF.Ovrd.tOvrdActivate(CLK:=FF.Ovrd.Active);
        FF.Ovrd.OvrdActLogAck S= FF.Ovrd.tOvrdActivate.Q;

        FF.Ovrd.tOvrdExpiring(CLK:=FF.Ovrd.Active);
        FF.Ovrd.OvrdExpLogAck S= FF.Ovrd.tOvrdExpiring.Q;

        FF.Ovrd.ElapsedTime := TIME_TO_UDINT(FF.Ovrd.Timer.ET);

        FF.Ovrd.RemainingTime := MAX(0, TO_DINT(FF.Ovrd.Timer.PT) - FF.Ovrd.ElapsedTime);

        // Clear pushbuttons
        FF.Ovrd.Activate := FALSE;
        FF.Ovrd.Deactivate := FALSE;

    END_IF
END_FOR
END_METHOD

{attribute 'obsolete' := 'Use EvaluateOverrides instead.'}
METHOD EvaluateVetos : BOOL
VAR_INPUT
END_VAR
END_METHOD

ACTION Execute:
EvaluateOverrides();
EvaluateOutput();
ExecuteLogging();
END_ACTION

{attribute 'no_check'}
METHOD ExecuteLogging : BOOL
VAR_INPUT
END_VAR
VAR
    FF : REFERENCE TO ST_FF;
    logIdx : DINT := 1;
END_VAR
VAR_INST
    HelloTimer : TOF := ( PT:=T#24h );
END_VAR

FOR logIdx := 1 to FF_ARRAY_UPPER_BOUND do

    FF REF= astFF[logIdx];

    IF NOT FF.Info.InUse THEN
        CONTINUE;
    ELSE
        IF FF.FaultAck THEN

            pmpsTypeCode := 1;
            FormulateLogJson(FF);
            fbLogger(sMsg := 'Fault, beam off', eSevr:=TcEventSeverity.Critical);

            FF.FaultAck := FALSE;
        END_IF

        IF FF.Ovrd.OvrdActLogAck THEN

            pmpsTypeCode := 2;
            FormulateLogJson(FF);

            fbLogger(sMsg := 'Override activated', eSevr:=TcEventSeverity.Warning);

            FF.Ovrd.OvrdActLogAck := FALSE;
        END_IF

        IF FF.Ovrd.OvrdExpLogAck THEN

            pmpsTypeCode := 3;
            FormulateLogJson(FF);

            fbLogger(sMsg := 'Override released', eSevr:=TcEventSeverity.Warning);

            FF.Ovrd.OvrdExpLogAck := FALSE;
        END_IF

        IF FF.ClearAck THEN

            pmpsTypeCode := 8;
            FormulateLogJson(FF);

            fbLogger(sMsg := 'Fault cleared', eSevr:=TcEventSeverity.Info);

            FF.ClearAck := FALSE;
        END_IF


    END_IF
END_FOR

// Log registration fault cleared
tFFRegFail(CLK:=xFastFaultRegFail);
IF tFFRegFail.Q THEN
    fbJson.StartObject();
    fbJson.AddKey('pmps_typecode');
    fbJson.AddUdint(5);
    fbJson.AddKey('pmps_path');
    fbJson.AddString(sPath);
    fbJson.EndObject();
    fbJson.CopyDocument(pDoc:=fbLogger.sJson, SIZEOF(fbLogger.sJson));
    fbLogger(sMsg := 'Fast fault registration failure cleared. This may be bad as a fast fault could go unoticed.',
        eSevr:=TcEventSeverity.Warning);
END_IF

// Say hello
HelloTimer.IN := NOT HelloTimer.Q;
HelloTimer();
IF HelloTimer.IN THEN
    pmpsTypeCode := 10;
    FormulateLogJson(FF);
    fbLogger(eSubsystem:=E_Subsystem.NILVALUE,
        eSevr := TcEventSeverity.Info,
        sMsg := 'FFO is alive');
    fbLogger.eSubsystem := E_Subsystem.MPS;
END_IF
END_METHOD

ACTION ExecuteNoLog:
EvaluateOverrides();
EvaluateOutput();
//ExecuteLogging();
END_ACTION

METHOD INTERNAL FormulateLogJson : STRING
VAR_INPUT
    FF : ST_FF;
END_VAR
fbJson.StartObject();
fbJson.AddKey('pmps_typecode');
fbJson.AddUdint(pmpsTypeCode);
fbJson.AddKey('pmps_path');
fbJson.AddString(FF.Info.sPath);
fbJson.AddKey('pmps_device_name');
fbJson.AddString(FF.Info.DevName);
fbJson.EndObject();
fbLogger.sJson := fbJson.GetDocument();
fbJson.ResetDocument();
END_METHOD

{attribute 'no_check'}
METHOD INTERNAL IdxCheckIn : BOOL
VAR_INPUT
    Idx : DINT;
    OK : BOOL;
    Reset : BOOL;
END_VAR
VAR
    stFF : ST_FF;
    BeamPermitted : BOOL;
END_VAR
Idx := LIMIT(1,Idx,FF_ARRAY_UPPER_BOUND);
stFF := THIS^.astFF[Idx];

// Updating internal fault state
stFF.OK := OK;

// Reset and latching logic
stFF.rtReset(CLK:=stFF.Reset (*epics*) OR Reset (*from other PLC logic *) );
stFF.Reset R= stFF.rtReset.Q;
stFF.bsFF(SET := stFF.rtReset.Q OR stFF.Info.AutoReset, RESET1:= NOT OK);

BeamPermitted := stFF.bsFF.Q1 OR stFF.Ovrd.Active OR ((i_xVeto OR CheckStoppers()) AND stFF.Info.Vetoable);

// Fault generation
IF NOT BeamPermitted THEN
    THIS^.xOK := FALSE; //Very clever, thanks Zach!
END_IF

// Fast fault accumulation
stFF.ftCountFault(CLK:=stFF.bsFF.Q1);
IF stFF.ftCountFault.Q THEN PMPS_GVL.AccumulatedFF := PMPS_GVL.AccumulatedFF + 1; END_IF

//Clear pushbuttons
stFF.Reset := FALSE;

// Log when this fault faults
stFF.FaultAck S= stFF.BeamPermitted AND NOT BeamPermitted;

// Log when this fault has cleared
stFF.ClearAck S= BeamPermitted AND NOT stFF.BeamPermitted;

stFF.BeamPermitted := BeamPermitted;

// Copy state back to ff struct
THIS^.astFF[Idx] := stFF;
END_METHOD

{attribute 'no_check'}
METHOD INTERNAL Register : BOOL
VAR_INPUT
    stFFInfo : ST_FFInfo := (
        sPath := '',
        Desc := '',
        TypeCode := 16#00,
        DevName := ''); // Fast fault information

END_VAR
VAR_OUTPUT
    FFOName : T_MaxString;
    Idx : UINT;
END_VAR
VAR
END_VAR
FFOName := THIS^.sPath;
Idx := THIS^.nIndex;

IF THIS^.nIndex <= FF_ARRAY_UPPER_BOUND THEN

    THIS^.astFF[MIN(THIS^.nIndex,FF_ARRAY_UPPER_BOUND)].Info:=stFFInfo;

    THIS^.nIndex := THIS^.nIndex + 1;

    Register := TRUE; // Add successful
ELSE
    fbJson.StartObject();
    fbJson.AddKey('pmps_typecode');
    fbJson.AddUdint(4);
    fbJson.AddKey('pmps_path');
    fbJson.AddString(stFFInfo.sPath);
    fbJson.AddKey('pmps_device_name');
    fbJson.AddString(stFFInfo.DevName);
    fbJson.EndObject();
    fbLogger.sJson := fbJson.GetDocument();
    fbJson.ResetDocument();
    fbLogger(sMsg:='Fast fault registration failed. Too many fast faults on this FFO.',
        eSevr:=TcEventSeverity.Warning,
        eSubsystem:=E_Subsystem.MPS);
    xFastFaultRegFail := TRUE;
    Register := FALSE; // Failed to add name to list
END_IF
END_METHOD

END_FUNCTION_BLOCK

// ---- HelperFunctions/F_SafeBPCompare.TcPOU
(*Compares BeamParam1 to BeamParam2: if the parameters of BeamParam1 are more conservative than BeamParam2
the result will be true. *)
// Does not consider status. Status must be evaluated elsewhere.
{attribute 'no_check'}
FUNCTION F_SafeBPCompare : BOOL
VAR_INPUT
    BeamParam1    :    ST_BeamParams; //Must be more conservative than 2
    BeamParam2    :    ST_BeamParams;
END_VAR
VAR
    // Internal Attenuation OK boolean
    xAttOK: BOOL := FALSE;
    // Internal Per-pulse energy OK boolean
    xPPmjOK: BOOL := FALSE;
    // Internal photon energy OK boolean
    xEvOK: BOOL := FALSE;
    // Internal Beam Rate OK boolean
    xRateOK: BOOL;
    //Internal Beam Class Range OK boolean
    xBCOK : BOOL := FALSE;
    idx : UINT;
    xAuxAttOK : BOOL := TRUE;
    xAuxAprtOK : BOOL := TRUE;

    Att1 : REFERENCE TO ST_PMPS_Attenuator;
    Att2 : REFERENCE TO ST_PMPS_Attenuator;

END_VAR


xAttOK := BeamParam1.nTran <= MIN(PMPS_GVL.TRANS_SCALING_FACTOR, (BeamParam2.nTran *(PMPS_GVL.TRANS_SCALING_FACTOR+PMPS_PARAM.TRANS_MARGIN))/PMPS_GVL.TRANS_SCALING_FACTOR );
xEvOK := (BeamParam1.neVRange AND BeamParam2.neVRange) = BeamParam1.neVRange;
xRateOK    := (BeamParam1.nRate <= BeamParam2.nRate) OR (PMPS_GVL.stCurrentBeamParameters.nMachineMode =1); //ignore in SC mode
xBCOK := ((BeamParam1.nBCRange AND BeamParam2.nBCRange) = BeamParam1.nBCRange) OR (PMPS_GVL.stCurrentBeamParameters.nMachineMode =0); //ignore in NC mode;

FOR idx:=1 to PMPS_GVL.AUX_ATTENUATORS DO
    Att1 REF= BeamParam1.astAttenuators[idx];
    Att2 REF= BeamParam2.astAttenuators[idx];
    xAuxAttOK R= ( Att1.nTran > MIN( PMPS_GVL.TRANS_SCALING_FACTOR, ( (Att2.nTran *(PMPS_GVL.TRANS_SCALING_FACTOR+PMPS_PARAM.TRANS_MARGIN))/PMPS_GVL.TRANS_SCALING_FACTOR ) ) );
END_FOR

FOR idx:=1 to PMPS_GVL.MAX_APERTURES DO
    xAuxAprtOK R= BeamParam1.astApertures[idx].Height > BeamParam2.astApertures[idx].Height OR
    BeamParam1.astApertures[idx].Width > BeamParam2.astApertures[idx].Width;
END_FOR

F_SafeBPCompare := xAttOK AND xEvOK AND xRateOK AND xAuxAprtOK AND xAuxAttOK AND xBCOK;

END_FUNCTION

// ---- HelperFunctions/F_ValidReqID.TcPOU
FUNCTION F_ValidReqID : BOOL
VAR_INPUT
    ReqID : DWORD;
END_VAR
VAR
END_VAR

F_ValidReqID := ReqID <> PMPS_GVL.EXCLUDED_ASSERTION_ID AND ReqID <> 0;

END_FUNCTION

// ---- HelperFunctions/F_SafeBPCompare0Rate.TcPOU
(*Compares BeamParam1 to BeamParam2: if the parameters of BeamParam1 are more conservative than BeamParam2
the result will be true. *)
(* When the Mode PV is in Cu 0-rate means this function will return true regardless of other conditions if the beam rate
is zero *)
(* When the Mode PV is in SC 0-bc means this function will return true regardless of other conditions if the beam class
is zero *)
FUNCTION F_SafeBPCompare0Rate : BOOL
VAR_INPUT
    BeamParam1    :    ST_BeamParams; //Must be more conservative than 2
    BeamParam2    :    ST_BeamParams;
END_VAR
VAR

    // Beam-rate is zero, masks all others considerations.
    xZeroRate: BOOL;
    //Beam class is zero i.e beam off, masks all other considerations.
    xZeroBC : BOOL;

END_VAR


xZeroRate  := (BeamParam1.nRate = 0) AND (PMPS_GVL.stCurrentBeamParameters.nMachineMode = 0);
xZeroBC  := (BeamParam1.nBCRange <= 1) AND (PMPS_GVL.stCurrentBeamParameters.nMachineMode =1);

F_SafeBPCompare0Rate := (xZeroRate OR xZeroBC) OR F_SafeBPCompare(BeamParam1, BeamParam2);

END_FUNCTION

// ---- HelperFunctions/FB_DummyArbIO.TcPOU
(* Use to test other library integrations of PMPS preemptive functionality *)
(* This block stands in for the FB_SubSysToArb_IO block. *)

FUNCTION_BLOCK FB_DummyArbIO IMPLEMENTS I_HigherAuthority, I_LowerAuthority
VAR_INPUT
    //stCurrentBP : REFERENCE TO ST_BeamParams; //Set to something to redirect currentBP update
    LA : I_LowerAuthority;

    tRateDelay : TIME; // Delay until rate is looped back into q_stSimulatedBPReadback
    tTransDelay : TIME; // Delay until transmission is looped back into q_stSimulatedBPReadback
    tPEDelay : TIME; // Delay until PE is looped back into q_stSimulatedBPReadback
    tAptDelay : TIME; // Delay until apertures are looped back into q_stSimulatedBPReadback
    tSattDelay : TIME; // Delay until apertures are looped back into q_stSimulatedBPReadback

END_VAR
VAR_OUTPUT
    q_stSimulatedBPReadback : ST_BeamParams; // Updated to
END_VAR
VAR_IN_OUT
    FFO : FB_HardwareFFOutput;
END_VAR
VAR
   bAutoUpdateBP : BOOL := FALSE; // Set by AutoUpdateBP property, if true causes this FB to update PMPS_GVL.stCurrentBP to the
   // requested value automatically within the RequestBP method and restore it within the RemoveRequest method
   stNewReqBP : ST_BeamParams;

   stReqOutBP : ST_BeamParams;// To be written on next ApplyBPReq call

   stSaveCurrentBP : ST_BeamParams; // Will be restored after RemoveRequest then ApplyBPReq call

   nSavedID : DWORD; // Used to simulate CheckRequest method

   tonRate : TON;
   tonTrans : TON;
   tonPE : TON;
   tonApt : TON;
   tonSatt : TON;
   tonBCRange: TON;
   tonBC :TON;

END_VAR


LA.ElevateRequest(THIS^);

ApplyBPReq(FALSE); //If autoupdate is set, this will propagate the request to PMPS_GVL.stCurrentBP;

